	//-------------------------------------------------------------------------------------------------------------------------------------------
	30:	//--- WriteParameter Vel_I AllSegments
		diResultSercosWriteServiceData 	:= SercosWriteServiceDataToAllSegments(	i_dwIDN					:= dwIDNCarrierVelI, 
																				i_dwDataStraightSegment	:= dwVelI_Straight, 
																				i_dwDataCurveSegment	:= dwVelI_Curve,
																				i_wMaxDataLength		:= 4);
		IF diResultSercosWriteServiceData = 0 THEN
			q_xWriteParameterDone	:= TRUE;
			diState	:= 40;
		ELSE
			q_xWriteParameterError	:= TRUE;
			diState	:= 1000;
		END_IF	
		
	//-------------------------------------------------------------------------------------------------------------------------------------------
	40: //--- WriteParameter TrackingDeviation WarningLevel AllSegments
		IF dwIDNDeviationLevelWarning > 0 THEN //--- value of 0 deactivate TrackingDeviation Detection
			diResultSercosWriteServiceData := SercosWriteServiceDataToAllSegments( 	i_dwIDN 				:= dwIDNDeviationLevelWarning,
																					i_dwDataStraightSegment	:= dwDeviationLevelWarning,
																					i_dwDataCurveSegment	:= dwDeviationLevelWarning,
																					i_wMaxDataLength 		:= 4);
		END_IF
		IF diResultSercosWriteServiceData = 0 THEN
			diState := 50;
		ELSE
			q_xWriteParameterError	:= TRUE;
			diState := 1000;
		END_IF

	//-------------------------------------------------------------------------------------------------------------------------------------------
	50: //--- WriteParameter TrackingDeviation ErrorLevel AllSegments
		IF dwIDNDeviationLevelError > 0 THEN //--- value of 0 deactivate TrackingDeviation Detection
			diResultSercosWriteServiceData := SercosWriteServiceDataToAllSegments( 	i_dwIDN 				:= dwIDNDeviationLevelError,
																					i_dwDataStraightSegment	:= dwDeviationLevelError,
																					i_dwDataCurveSegment	:= dwDeviationLevelError,
																					i_wMaxDataLength 		:= 4);
		END_IF
		IF diResultSercosWriteServiceData = 0 THEN
			diState := 60;
		ELSE
			q_xWriteParameterError	:= TRUE;
			diState := 1000;
		END_IF		
		
	//-------------------------------------------------------------------------------------------------------------------------------------------
	60:	//--- WriteParameter: Maximum Current AllSegments
		diResultSercosWriteServiceData 	:= SercosWriteServiceDataToAllSegments(	i_dwIDN					:= dwIDNCarrierMaxcurr, 
																				i_dwDataStraightSegment	:= dwMaxCurr, 
																				i_dwDataCurveSegment	:= dwMaxCurr,
																				i_wMaxDataLength		:= 2);
		IF diResultSercosWriteServiceData = 0 THEN
			diState := 70;
		ELSE
			q_xWriteParameterError	:= TRUE;
			diState	:= 1000;
		END_IF	
	
	//-------------------------------------------------------------------------------------------------------------------------------------------
	70:	//--- WriteParameter: Load of Carrier AllSegments
		diResultSercosWriteServiceData 	:= SercosWriteServiceDataToAllSegments(	i_dwIDN					:= dwIDNCarrierLoad, 
																				i_dwDataStraightSegment	:= dwMaxload, 
																				i_dwDataCurveSegment	:= dwMaxload, 
																				i_wMaxDataLength		:= 4);
		IF diResultSercosWriteServiceData = 0 THEN
			q_xWriteParameterDone	:= TRUE;
			diState := 0;
		ELSE
			q_xWriteParameterError	:= TRUE;
			diState	:= 1000;
		END_IF	
	
	//-------------------------------------------------------------------------------------------------------------------------------------------
	1000: //--- ErrorState
		;
	
END_CASE

METHOD SercosWriteServiceDataToAllSegments : DINT
VAR_INPUT
	i_dwIDN					: DWORD;
	i_dwDataCurveSegment	: DWORD;	
	i_dwDataStraightSegment	: DWORD;	
	i_wMaxDataLength		: WORD;
END_VAR
VAR
	udiIndex				: UDINT;
END_VAR
FOR udiIndex := 1  TO GVL_MulticarrierConfiguration.Gc_astTracks[1].udiNumberOfSegments DO
	

    IF GVL_MulticarrierConfiguration.Gc_astSegmentTypes[GVL_MulticarrierConfiguration.Gc_astTracks[1].astSegments[udiIndex].diSegmentTypesIndex].xIsCurved  
    THEN        
        SercosWriteServiceDataToAllSegments := SystemInterface.FC_SercosWriteServiceDataByTopAddr(    
                                                                    i_wTopoAddr         := TO_WORD(udiIndex), 
                                                                    i_dwIDN             := i_dwIDN,
                                                                    i_wType             := 5,
                                                                    i_dwPointerToData   := ADR(i_dwDataCurveSegment),
                                                                    i_wMaxDataLen       := i_wMaxDataLength);
    ELSE
        SercosWriteServiceDataToAllSegments := SystemInterface.FC_SercosWriteServiceDataByTopAddr(    
                                                                    i_wTopoAddr         := TO_WORD(udiIndex), 
                                                                    i_dwIDN             := i_dwIDN,
                                                                    i_wType             := 5,
                                                                    i_dwPointerToData   := ADR(i_dwDataStraightSegment),
                                                                    i_wMaxDataLen       := i_wMaxDataLength);
    END_IF    

    IF SercosWriteServiceDataToAllSegments <> 0 THEN
        RETURN;
    END_IF
END_FOR
END_METHOD

METHOD StartAndSetParameter
VAR_INPUT
	i_dwPosP_Straight				: DWORD;
	i_dwVelP_Straight				: DWORD;
	i_dwVelI_Straight				: DWORD;  
	i_dwPosP_Curve					: DWORD;
	i_dwVelP_Curve					: DWORD;
	i_dwVelI_Curve					: DWORD;  
	i_dwMaxCurr			            : DWORD;
    i_dwMaxload					    : DWORD;
    i_dwDeviationLevelWarning       : DWORD;
    i_dwDeviationLevelError         : DWORD;
	
	
	
END_VAR
dwPosP_Straight	:= 	i_dwPosP_Straight;
dwVelP_Straight	:=	i_dwVelP_Straight;
dwVelI_Straight	:=	i_dwVelI_Straight;

dwPosP_Curve	:= 	i_dwPosP_Curve;
dwVelP_Curve	:=	i_dwVelP_Curve;
dwVelI_Curve	:=	i_dwVelI_Curve;

dwMaxCurr			      := i_dwMaxCurr;
dwMaxload				  := i_dwMaxload;
dwDeviationLevelWarning   := i_dwDeviationLevelWarning;
dwDeviationLevelError     := i_dwDeviationLevelError;

xStart 		:=  TRUE;
END_METHOD

END_PROGRAM

// LMC_PacDrive/Application/TemplateFullProgrammingFramework/TaskCalls/SR_Diagnostics
PROGRAM SR_Diagnostics

VAR
	fbDiagnosticsManager : TPL.FB_DiagnosticsManager;
	stComStructure 		 : TPL.ST_DiagnosticsManagerToDiagSource;
	
	stWarning 		: TPL.ST_Exception;
	etLastDiagExt	: TPL.ET_DiagExt := TPL.ET_DiagExt.Ok;

	(* Add the instances of your sources for diag data here *)
	fbTemplateStaticStructureDiagSource	: TPL.FB_TemplateStaticStructureDiagSource;
	fbExceptionListDiagSource			: TPL.FB_ExceptionListDiagSource;
	fbExceptionDelayListDiagSource		: TPL.FB_ExceptionDelayListDiagSource;
	fbLogDataListDiagSource				: TPL.FB_LogDataListDiagSource;	
	fbAxisModuleDiagSource				: AXM.FB_AxisModuleDiagSource;
	xPrintCamData						: BOOL := TRUE;
	fbApplicationLoggerDiagSource		: FB_ApplicationLoggerDiagSource;

	(* example diag sources *)
	fbExampleTableDiagSource			: FB_ExampleTableDiagSource;
	fbExampleTreeDiagSource				: FB_ExampleTreeDiagSource;
END_VAR

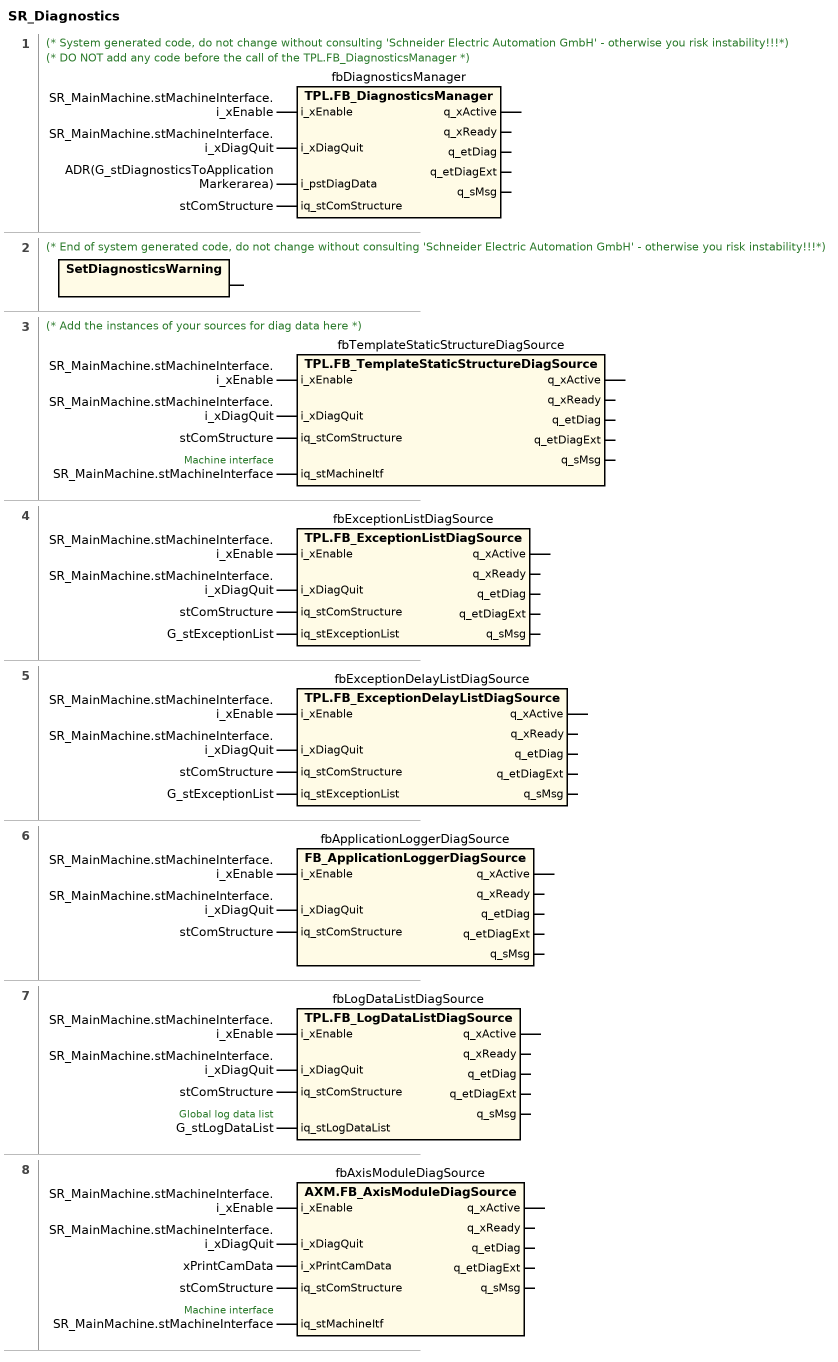
// NETWORK 1
// (* System generated code, do not change without consulting 'Schneider Electric Automation GmbH' - otherwise you risk instability!!!*)
// (* DO NOT add any code before the call of the TPL.FB_DiagnosticsManager *)
fbDiagnosticsManager(
    i_xEnable := SR_MainMachine.stMachineInterface.i_xEnable,
    i_xDiagQuit := SR_MainMachine.stMachineInterface.i_xDiagQuit,
    i_pstDiagData := ADR(G_stDiagnosticsToApplicationMarkerarea),
    iq_stComStructure := stComStructure); // TPL.FB_DiagnosticsManager

// NETWORK 2
// (* End of system generated code, do not change without consulting 'Schneider Electric Automation GmbH' - otherwise you risk instability!!!*)
SetDiagnosticsWarning();

// NETWORK 3
// (* Add the instances of your sources for diag data here *)
//   fbTemplateStaticStructureDiagSource: Add the instances of your sources for diag data here
//   SR_MainMachine.stMachineInterface: Machine interface
fbTemplateStaticStructureDiagSource(
    i_xEnable := SR_MainMachine.stMachineInterface.i_xEnable,
    i_xDiagQuit := SR_MainMachine.stMachineInterface.i_xDiagQuit,
    iq_stComStructure := stComStructure,
    iq_stMachineItf := SR_MainMachine.stMachineInterface); // TPL.FB_TemplateStaticStructureDiagSource

// NETWORK 4
fbExceptionListDiagSource(
    i_xEnable := SR_MainMachine.stMachineInterface.i_xEnable,
    i_xDiagQuit := SR_MainMachine.stMachineInterface.i_xDiagQuit,
    iq_stComStructure := stComStructure,
    iq_stExceptionList := G_stExceptionList); // TPL.FB_ExceptionListDiagSource

// NETWORK 5
fbExceptionDelayListDiagSource(
    i_xEnable := SR_MainMachine.stMachineInterface.i_xEnable,
    i_xDiagQuit := SR_MainMachine.stMachineInterface.i_xDiagQuit,
    iq_stComStructure := stComStructure,
    iq_stExceptionList := G_stExceptionList); // TPL.FB_ExceptionDelayListDiagSource

// NETWORK 6
fbApplicationLoggerDiagSource(
    i_xEnable := SR_MainMachine.stMachineInterface.i_xEnable,
    i_xDiagQuit := SR_MainMachine.stMachineInterface.i_xDiagQuit,
    iq_stComStructure := stComStructure); // FB_ApplicationLoggerDiagSource

// NETWORK 7
//   G_stLogDataList: Global log data list
fbLogDataListDiagSource(
    i_xEnable := SR_MainMachine.stMachineInterface.i_xEnable,
    i_xDiagQuit := SR_MainMachine.stMachineInterface.i_xDiagQuit,
    iq_stComStructure := stComStructure,
    iq_stLogDataList := G_stLogDataList); // TPL.FB_LogDataListDiagSource

// NETWORK 8
//   SR_MainMachine.stMachineInterface: Machine interface
fbAxisModuleDiagSource(
    i_xEnable := SR_MainMachine.stMachineInterface.i_xEnable,
    i_xDiagQuit := SR_MainMachine.stMachineInterface.i_xDiagQuit,
    i_xPrintCamData := xPrintCamData,
    iq_stComStructure := stComStructure,
    iq_stMachineItf := SR_MainMachine.stMachineInterface); // AXM.FB_AxisModuleDiagSource

ACTION SetDiagnosticsWarning:
(* System generated code, do not change without consulting 'Schneider Electric Automation GmbH' - otherwise you risk instability!!!*)
						
(* Signal exception during diagnostics, but as diagnostics should not influence the machine, create only a warning *)
IF(fbDiagnosticsManager.q_etDiag <> GD.ET_Diag.Ok AND fbDiagnosticsManager.q_etDiagExt <> etLastDiagExt) THEN
	
	stWarning.etDiag		:= GD.ET_Diag.DiagActive;
	stWarning.udiDiagExt	:= ET_DiagExt.DiagnosticsWarning;
	stWarning.sDiagExt		:= FC_EtDiagExtToString(stWarning.udiDiagExt);
	stWarning.udiModuleId	:= SR_MainMachine.c_udiMainModuleId;
	stWarning.sMsg			:= CONCAT(CONCAT('SR_Diagnostics: ', GD.FC_EtDiagToString(fbDiagnosticsManager.q_etDiag)), CONCAT(' ; ', TPL.FC_EtDiagExtToString(fbDiagnosticsManager.q_etDiagExt)));
	stWarning.sModuleName	:= SR_MainMachine.stMachineInterface.i_sModuleName;
	stWarning.etSource		:= TPL.ET_ExceptionSource.Logger;
	
	TPL.FC_SetException(i_xExceptionActive	:= TRUE,
						iq_stException		:= stWarning,
						iq_stExceptionList	:= G_stExceptionList,
						iq_stLogDataList	:= G_stLogDataList);
END_IF

etLastDiagExt := fbDiagnosticsManager.q_etDiagExt;
(* End of system generated code, do not change without consulting 'Schneider Electric Automation GmbH' - otherwise you risk instability!!!*)
END_ACTION

END_PROGRAM

// LMC_PacDrive/Application/TemplateFullProgrammingFramework/Examples/ExampleDiagSources/FB_ApplicationLoggerDiagSource
FUNCTION_BLOCK PUBLIC FB_ApplicationLoggerDiagSource
VAR_INPUT
	i_xEnable			: BOOL;
	i_xDiagQuit			: BOOL;
END_VAR

VAR_IN_OUT
	iq_stComStructure	: TPL.ST_DiagnosticsManagerToDiagSource;
END_VAR

VAR_OUTPUT
	q_xActive			: BOOL;
	q_xReady			: BOOL;
	q_etDiag			: GD.ET_Diag := GD.ET_Diag.Ok;
	q_etDiagExt			: ET_DiagExt := ET_DiagExt.Disabled;
	q_sMsg				: STRING[80];
END_VAR

VAR
	xEnableFlag		: BOOL;
	diState			: DINT;

	udiOwnSourceId	: UDINT := 0;

	fbTreeWriter	: TPL.FB_TreeWriter;
	
	diOldCmd		: DINT := 0;
	diCmdExecState	: DINT := 0;

	etDiagBuffer		: GD.ET_Diag;
	etDiagExtBufferTPL	: TPL.ET_DiagExt;
	etDiagExtBufferAPL	: APL.ET_DiagExt;
	sMsgBuffer			: STRING[80];
	
	rtrigDiagQuit	: Standard.R_TRIG;
	
	fbAppLogHandler			: APL.FB_ApplicationLoggerHandler;
	stLogEntry				: APL.ST_LogEntry;
	ifLoggerPoint			: APL.IF_LoggerPoint;
	udiLogEntryCount		: UDINT;
	udiLogEntryCountMax		: UDINT;
	udiLogEntryId			: UDINT;
	udiLoggerPointCount		: UDINT;
	udiLoggerPointCountMax	: UDINT;
END_VAR

VAR CONSTANT
	c_sName			: STRING[TPL.Gc_udiTableWriterMaxNameLength] := 'ApplicationLogger';
	c_sTypeName		: STRING[TPL.Gc_udiTableWriterMaxNameLength] := 'APL_';
END_VAR

IF i_xEnable AND NOT xEnableFlag THEN
	xEnableFlag := TRUE;
	q_xActive := TRUE;
	SetDiagOutputs(	i_etDiag	:= GD.ET_Diag.Ok,
					i_etDiagExt	:= ET_DiagExt.WaitUntilDiagnosticsManagerReady,
					i_sMsg		:= '');	
	diState := 10;
	
ELSIF NOT i_xEnable AND xEnableFlag THEN
	xEnableFlag := FALSE;
	IF udiOwnSourceId <> 0 THEN		
		SetDiagOutputs(	i_etDiag	:= GD.ET_Diag.Ok,
						i_etDiagExt	:= ET_DiagExt.WaitUntilDisabled,
						i_sMsg		:= '');
		diState := 100;
	ELSIF udiOwnSourceId = 0 THEN		
		SetDiagOutputs(	i_etDiag	:= GD.ET_Diag.Ok,
						i_etDiagExt	:= ET_DiagExt.Disabled,
						i_sMsg		:= '');
	END_IF
END_IF

DiagQuit();

CASE diState OF
	
	0:	(* Disable & exception state *)
		;
	
	10:	(* Wait until diagnostics manager ready *)
		IF iq_stComStructure.i_xDiagnosticsManagerReady THEN
			SetDiagOutputs(	i_etDiag	:= GD.ET_Diag.Ok,
							i_etDiagExt	:= ET_DiagExt.WaitUntilDiagSourceRegistered,
							i_sMsg		:= '');
			diState := 20;
		END_IF

	20:	(* Wait until diag source registered *)	
		IF NOT iq_stComStructure.i_xDiagnosticsManagerReady THEN
			SetDiagOutputs(	i_etDiag	:= GD.ET_Diag.Ok,
							i_etDiagExt	:= ET_DiagExt.WaitUntilDiagnosticsManagerReady,
							i_sMsg		:= '');	
			diState := 10;
	
		(* only write to register structure if no one else has done it in this cylce *)
		ELSIF (NOT iq_stComStructure.iq_stRegister.xUsed AND iq_stComStructure.iq_stRegister.udiNextId <> 0) THEN
			(* register *)
			iq_stComStructure.iq_stRegister.xUsed := TRUE;
			iq_stComStructure.iq_stRegister.sName		:= c_sName;
			iq_stComStructure.iq_stRegister.sTypeName	:= c_sTypeName;
			udiOwnSourceId := iq_stComStructure.iq_stRegister.udiNextId; (* register with this id; required for the following communication *)
			
			q_xReady := TRUE;
			SetDiagOutputs(	i_etDiag	:= GD.ET_Diag.Ok,
							i_etDiagExt	:= ET_DiagExt.WaitForCommunication,
							i_sMsg		:= '');
			diState := 30;
		END_IF
	
	30:	(* Wait for communication *)	
		IF NOT iq_stComStructure.i_xDiagnosticsManagerReady THEN

			CancelWriting();
									
			udiOwnSourceId	:= 0;
			
			SetDiagOutputs(	i_etDiag	:= GD.ET_Diag.Ok,
							i_etDiagExt	:= ET_DiagExt.WaitUntilDiagnosticsManagerReady,
							i_sMsg		:= '');	
			diState := 10;
			RETURN;
			
		ELSIF (iq_stComStructure.i_udiComWithId = udiOwnSourceId) THEN		(* Am I adressed? *)
			
			WriteDiagDataControl();

		ELSE
			iq_stComStructure.q_lrProgress := 0.0;
			
			CancelWriting();
						
			SetDiagOutputs(	i_etDiag	:= GD.ET_Diag.Ok,
							i_etDiagExt	:= ET_DiagExt.WaitForCommunication,
							i_sMsg		:= '');
		END_IF
		
	100: (* Wait until disabled *)	
		IF NOT iq_stComStructure.i_xDiagnosticsManagerReady THEN

			CancelWriting();
									
			udiOwnSourceId	:= 0;
			
			SetDiagOutputs(	i_etDiag	:= GD.ET_Diag.Ok,
							i_etDiagExt	:= ET_DiagExt.Disabled,
							i_sMsg		:= '');	
	
		ELSIF (iq_stComStructure.i_udiComWithId = udiOwnSourceId) THEN		(* Am I adressed? *)
			
			WriteDiagDataControl();
			
		(* only write to register structure if no one else has done it in this cylce *)
		ELSIF (NOT iq_stComStructure.iq_stRegister.xUsed AND NOT iq_stComStructure.iq_stRegister.xUnsubscribe) AND 
			   NOT iq_stComStructure.i_xDiagnosticsActive THEN
			   
			iq_stComStructure.iq_stRegister.xUsed			:= TRUE;
			
			iq_stComStructure.iq_stRegister.xUnsubscribe	:= TRUE;
			iq_stComStructure.iq_stRegister.udiSourceId		:= udiOwnSourceId;
			
			q_xActive := FALSE;
			
			SetDiagOutputs(	i_etDiag	:= GD.ET_Diag.Ok,
							i_etDiagExt	:= ET_DiagExt.Disabled,
							i_sMsg		:= '');
		END_IF
END_CASE

IF q_xReady THEN	
	IF(diCmdExecState <> 0) THEN
		WriteDiagDataToFile();
		
		IF(iq_stComStructure.iq_diCmd <= 0) THEN
			diOldCmd := iq_stComStructure.iq_diCmd;
		END_IF
	END_IF	
END_IF

METHOD INTERNAL CancelWriting
VAR_INPUT
END_VAR
(* Deactivate writing if we are (for whatever reason) no longer adressed.
   May happen in case network connection with Diagnostics is disrupted or Source will be disabled *)

THIS^.diOldCmd			:= 0;
THIS^.diCmdExecState	:= 0;
END_METHOD

METHOD INTERNAL DiagQuit
VAR_INPUT
END_VAR
IF THIS^.i_xEnable AND THIS^.q_xActive AND THIS^.q_etDiag <> GD.ET_Diag.Ok AND THIS^.diState = 0 THEN

	THIS^.rtrigDiagQuit(CLK := THIS^.i_xDiagQuit);
	IF THIS^.rtrigDiagQuit.Q THEN
		CancelWriting();
									
		THIS^.udiOwnSourceId	:= 0;
		
		THIS^.fbTreeWriter.FB_Init(bInitRetains := FALSE, bInCopyCode := FALSE);
			
		THIS^.q_xReady		:= TRUE;
		THIS^.q_etDiag		:= GD.ET_Diag.Ok;
		THIS^.q_etDiagExt	:= ET_DiagExt.WaitUntilDiagnosticsManagerReady;
		THIS^.q_sMsg		:= '';
	
		THIS^.diState := 10;
	END_IF

END_IF
END_METHOD

METHOD INTERNAL ExceptionDuringWriting : BOOL
VAR_INPUT
END_VAR
(* exception during writing *)
CASE THIS^.etDiagExtBufferTPL OF
	TPL.ET_DiagExt.TreeStartAlreadySuccessfullyCalled,		// FB_TreeWriter.TreeStart	
	TPL.ET_DiagExt.FileIdNotSet,							// FB_TreeWriter.TreeStart							
	TPL.ET_DiagExt.FileIdInvalid,							// FB_TreeWriter.TreeStart & FB_TreeWriter.NodeStart & FB_TreeWriter.Parameter & FB_TreeWriter.NodeEnd & FB_TreeWriter.TreeEnd								
	TPL.ET_DiagExt.FileNotOpen,								// FB_TreeWriter.TreeStart & FB_TreeWriter.NodeStart & FB_TreeWriter.Parameter & FB_TreeWriter.NodeEnd & FB_TreeWriter.TreeEnd								
	TPL.ET_DiagExt.UnexpectedFeedback,						// FB_TreeWriter.TreeStart & FB_TreeWriter.NodeStart & FB_TreeWriter.Parameter & FB_TreeWriter.NodeEnd & FB_TreeWriter.TreeEnd								
	TPL.ET_DiagExt.TreeStartNotCalled,						// FB_TreeWriter.NodeStart								
	TPL.ET_DiagExt.TreeStartNotSuccessfullyCalled,			// FB_TreeWriter.NodeStart								
	TPL.ET_DiagExt.NoMoreNodeOpen,							// FB_TreeWriter.Parameter & FB_TreeWriter.NodeEnd						
	TPL.ET_DiagExt.CallTreeStartFirst,						// FB_TreeWriter.TreeEnd								
	TPL.ET_DiagExt.NodesStillOpen:							// FB_TreeWriter.TreeEnd	
	
		SetDiagOutputs(	i_etDiag	:= GD.ET_Diag.UnexpectedProgramBehavior,
						i_etDiagExt	:= ET_DiagExt.UnexpectedFeedback,
						i_sMsg		:= PDL.FC_MultiConcat(	i_sString1	:= 'FB_TreeWriter: ', 
															i_sString2	:= GD.FC_EtDiagToString(THIS^.etDiagBuffer), 
															i_sString3	:= ' - ', 
															i_sString4	:= TPL.FC_EtDiagExtToString(THIS^.etDiagExtBufferTPL), 
															q_etDiag	=> , 
															q_etDiagExt	=> )); 								
	ELSE
		SetDiagOutputs(	i_etDiag	:= GD.ET_Diag.UnexpectedProgramBehavior,
						i_etDiagExt	:= ET_DiagExt.UnexpectedFeedback,
						i_sMsg		:= PDL.FC_MultiConcat(	i_sString1	:= 'FB_TreeWriter: ', 
															i_sString2	:= GD.FC_EtDiagToString(THIS^.etDiagBuffer), 
															i_sString3	:= ' - ', 
															i_sString4	:= TPL.FC_EtDiagExtToString(THIS^.etDiagExtBufferTPL), 
															q_etDiag	=> , 
															q_etDiagExt	=> )); 						
END_CASE
		
CancelWriting();
END_METHOD

METHOD INTERNAL SetDiagOutputs : BOOL
VAR_INPUT
	i_etDiag		: GD.ET_Diag;
	i_etDiagExt		: ET_DiagExt;
	i_sMsg			: STRING[80];
END_VAR
IF THIS^.q_etDiag = GD.ET_Diag.Ok OR i_etDiagExt = ET_DiagExt.Disabled THEN

	IF i_etDiag <> GD.ET_Diag.Ok OR i_etDiagExt = ET_DiagExt.Disabled THEN
		
		IF i_etDiag <> GD.ET_Diag.Ok THEN
			THIS^.iq_stComStructure.iq_diCmd := -THIS^.iq_stComStructure.iq_diCmd;
		END_IF
		
		IF i_etDiagExt = ET_DiagExt.Disabled THEN
			THIS^.q_xActive := FALSE;
			
			CancelWriting();
		END_IF
		
		THIS^.q_xReady := FALSE;
		THIS^.diState := 0;
	END_IF
	
	THIS^.q_etDiag		:= i_etDiag;
	THIS^.q_etDiagExt	:= i_etDiagExt;
	THIS^.q_sMsg		:= i_sMsg;
END_IF
END_METHOD

METHOD INTERNAL WriteDiagDataControl : BOOL
VAR_INPUT
END_VAR
IF (THIS^.diOldCmd <> THIS^.iq_stComStructure.iq_diCmd AND THIS^.iq_stComStructure.iq_diCmd > 0) THEN
	THIS^.diOldCmd := THIS^.iq_stComStructure.iq_diCmd;
	
	(* new command, start execution *)
	IF THIS^.iq_stComStructure.iq_diCmd = 1 THEN
		IF (THIS^.iq_stComStructure.i_diFileId > 0) THEN
			SetDiagOutputs(	i_etDiag		:= GD.ET_Diag.Ok,
							i_etDiagExt		:= ET_DiagExt.WritingToFile,
							i_sMsg			:= '');
			THIS^.iq_stComStructure.q_lrProgress := 0.0;
			THIS^.fbTreeWriter.diFileId := THIS^.iq_stComStructure.i_diFileId;
			THIS^.diCmdExecState := 1; (* start writing to file *)
		ELSE
			(* invalid file id *)
			SetDiagOutputs(	i_etDiag		:= GD.ET_Diag.InputParameterInvalid,
							i_etDiagExt		:= ET_DiagExt.FileIdInvalid,
							i_sMsg			:= CONCAT('Invalid file Id iq_stComStructure.i_diFileId: ', DINT_TO_STRING(THIS^.iq_stComStructure.i_diFileId)));
		END_IF
	ELSE
		(* unkown cmd *)
		SetDiagOutputs(	i_etDiag		:= GD.ET_Diag.InputParameterInvalid,
						i_etDiagExt		:= ET_DiagExt.CmdUnknown,
						i_sMsg			:= CONCAT('Unknown command iq_stComStructure.diCmd: ', DINT_TO_STRING(THIS^.iq_stComStructure.iq_diCmd)));

		CancelWriting();
	END_IF
END_IF
END_METHOD

METHOD WriteDiagDataToFile
VAR_INPUT
END_VAR
TPL.FC_CanContinueWriting(iq_stCanContinueWriting := THIS^.iq_stComStructure.iq_stCanContinueWriting); (* loop as long as we can continue to write *)

WHILE (THIS^.iq_stComStructure.iq_stCanContinueWriting.xCanContinue) DO
	
	CASE THIS^.diCmdExecState OF
		1:	(* start writing *)
			THIS^.fbTreeWriter.TreeStart(	i_sName					:= THIS^.c_sName, 
											i_sTypeName				:= THIS^.c_sTypeName, 
											i_sTitleEnglish			:= 'ApplicationLogger', 
											i_sTitleGerman			:= 'ApplicationLogger', 
											i_uiPrintRank			:= 14, 
											i_sEmptyListTextEnglish	:= 'No data available to show', 
											i_sEmptyListTextGerman	:= 'Keine Daten zum Anzeigen vorhanden',
											q_etDiag				=> THIS^.etDiagBuffer,
											q_etDiagExt				=> THIS^.etDiagExtBufferTPL,
											q_sMsg					=> THIS^.sMsgBuffer);
			IF THIS^.etDiagBuffer <> GD.ET_Diag.Ok THEN
				ExceptionDuringWriting();
				EXIT;
			END_IF
			THIS^.diCmdExecState := 50;

		50:	(* Start LogEntryList *)
			THIS^.fbTreeWriter.NodeStart(	i_sName		:= 'LogEntry list',
											q_etDiag	=> etDiagBuffer,
											q_etDiagExt	=> etDiagExtBufferTPL,
											q_sMsg		=> sMsgBuffer);
			IF THIS^.etDiagBuffer <> GD.ET_Diag.Ok THEN
				ExceptionDuringWriting();
				EXIT;
			END_IF
			THIS^.udiLogEntryCount := 1;
			THIS^.udiLogEntryCountMax := 50;
			THIS^.udiLogEntryId := THIS^.fbAppLogHandler.udiFirstLogEntryId;
			THIS^.diCmdExecState := 51;
			
		51: (* write LogEntrys *)
			WHILE (THIS^.udiLogEntryCount < THIS^.udiLogEntryCountMax) AND (THIS^.udiLogEntryCount <= THIS^.fbAppLogHandler.udiNumberOfLogEntries) DO
				THIS^.fbTreeWriter.NodeStart(	i_sName		:= UDINT_TO_STRING(THIS^.udiLogEntryId),
												q_etDiag	=> etDiagBuffer,
												q_etDiagExt	=> etDiagExtBufferTPL,
												q_sMsg		=> sMsgBuffer);
				IF THIS^.etDiagBuffer <> GD.ET_Diag.Ok THEN
					ExceptionDuringWriting();
					RETURN;
				END_IF					

					THIS^.fbAppLogHandler.GetLogEntry(	i_udiId			:= THIS^.udiLogEntryId,
														q_stLogEntry	=> THIS^.stLogEntry,
														q_etDiag		=> THIS^.etDiagBuffer,
														q_etDiagExt		=> THIS^.etDiagExtBufferAPL);
					IF (THIS^.etDiagBuffer <> GD.ET_Diag.Ok) THEN
						ExceptionDuringWriting();
						RETURN;
					END_IF
				
					THIS^.fbTreeWriter.Parameter(	i_sName		:= 'udiId', 
													i_sValue	:= UDINT_TO_STRING(THIS^.stLogEntry.udiId),
													q_etDiag	=> etDiagBuffer,
													q_etDiagExt	=> etDiagExtBufferTPL,
													q_sMsg		=> sMsgBuffer);
					IF etDiagBuffer <> GD.ET_Diag.Ok THEN
						ExceptionDuringWriting();
						RETURN;
					END_IF

					THIS^.fbTreeWriter.Parameter(	i_sName		:= 'udiLoggerPointId', 
													i_sValue	:= UDINT_TO_STRING(THIS^.stLogEntry.udiLoggerPointId),
													q_etDiag	=> etDiagBuffer,
													q_etDiagExt	=> etDiagExtBufferTPL,
													q_sMsg		=> sMsgBuffer);
					IF etDiagBuffer <> GD.ET_Diag.Ok THEN
						ExceptionDuringWriting();
						RETURN;
					END_IF
					THIS^.fbTreeWriter.Parameter(	i_sName		:= 'sMessage', 
													i_sValue	:= THIS^.stLogEntry.sMessage,
													q_etDiag	=> etDiagBuffer,
													q_etDiagExt	=> etDiagExtBufferTPL,
													q_sMsg		=> sMsgBuffer);
					IF etDiagBuffer <> GD.ET_Diag.Ok THEN
						ExceptionDuringWriting();
						RETURN;
					END_IF
					THIS^.fbTreeWriter.Parameter(	i_sName		:= 'etDiag', 
													i_sValue	:= GD.FC_EtDiagToString(i_etDiag := THIS^.stLogEntry.etDiag),
													q_etDiag	=> etDiagBuffer,
													q_etDiagExt	=> etDiagExtBufferTPL,
													q_sMsg		=> sMsgBuffer);
					IF etDiagBuffer <> GD.ET_Diag.Ok THEN
						ExceptionDuringWriting();
						RETURN;
					END_IF
					THIS^.fbTreeWriter.Parameter(	i_sName		:= 'udiDiagExt', 
													i_sValue	:= UDINT_TO_STRING(THIS^.stLogEntry.udiDiagExt),
													q_etDiag	=> etDiagBuffer,
													q_etDiagExt	=> etDiagExtBufferTPL,
													q_sMsg		=> sMsgBuffer);
					IF etDiagBuffer <> GD.ET_Diag.Ok THEN
						ExceptionDuringWriting();
						RETURN;
					END_IF
					THIS^.fbTreeWriter.Parameter(	i_sName		:= 'dtDate', 
													i_sValue	:= DATE_TO_STRING(THIS^.stLogEntry.dtDate),
													q_etDiag	=> etDiagBuffer,
													q_etDiagExt	=> etDiagExtBufferTPL,
													q_sMsg		=> sMsgBuffer);
					IF etDiagBuffer <> GD.ET_Diag.Ok THEN
						ExceptionDuringWriting();
						RETURN;
					END_IF
					THIS^.fbTreeWriter.Parameter(	i_sName		:= 'todTime', 
													i_sValue	:= TOD_TO_STRING(THIS^.stLogEntry.todTime),
													q_etDiag	=> etDiagBuffer,
													q_etDiagExt	=> etDiagExtBufferTPL,
													q_sMsg		=> sMsgBuffer);
					IF etDiagBuffer <> GD.ET_Diag.Ok THEN
						ExceptionDuringWriting();
						RETURN;
					END_IF
					THIS^.fbTreeWriter.Parameter(	i_sName		:= 'etLogLevel', 
													i_sValue	:= APL.FC_EtLogLevelToString(i_etLogLevel := THIS^.stLogEntry.etLogLevel),
													q_etDiag	=> etDiagBuffer,
													q_etDiagExt	=> etDiagExtBufferTPL,
													q_sMsg		=> sMsgBuffer);
					IF etDiagBuffer <> GD.ET_Diag.Ok THEN
						ExceptionDuringWriting();
						RETURN;
					END_IF
					
				THIS^.fbTreeWriter.NodeEnd(	q_etDiag	=> etDiagBuffer,
											q_etDiagExt	=> etDiagExtBufferTPL,
											q_sMsg		=> sMsgBuffer);	
				IF THIS^.etDiagBuffer <> GD.ET_Diag.Ok THEN
					ExceptionDuringWriting();
					RETURN;
				END_IF	
			
				THIS^.udiLogEntryCount := THIS^.udiLogEntryCount +1;
				THIS^.udiLogEntryId := THIS^.udiLogEntryId +1;
			END_WHILE
			THIS^.udiLogEntryCountMax := THIS^.udiLogEntryCountMax + 50;
			IF (THIS^.udiLogEntryCount > THIS^.fbAppLogHandler.udiNumberOfLogEntries) THEN
				THIS^.fbTreeWriter.NodeEnd(	q_etDiag	=> etDiagBuffer,
											q_etDiagExt	=> etDiagExtBufferTPL,
											q_sMsg		=> sMsgBuffer);	
				IF THIS^.etDiagBuffer <> GD.ET_Diag.Ok THEN
					ExceptionDuringWriting();
					EXIT;
				END_IF
				THIS^.diCmdExecState := 60;
			END_IF
		
		60: (* Start LoggerPoint list *)
			THIS^.fbTreeWriter.NodeStart(	i_sName		:= 'LoggerPoint list',
											q_etDiag	=> etDiagBuffer,
											q_etDiagExt	=> etDiagExtBufferTPL,
											q_sMsg		=> sMsgBuffer);
			IF THIS^.etDiagBuffer <> GD.ET_Diag.Ok THEN
				ExceptionDuringWriting();
				EXIT;
			END_IF
			THIS^.udiLoggerPointCount := 1;
			THIS^.udiLoggerPointCountMax := 50;
			THIS^.diCmdExecState := 61;	
			
		61: (* write LoggerPoint list *)
			WHILE (THIS^.udiLoggerPointCount < THIS^.udiLoggerPointCountMax) AND (THIS^.udiLoggerPointCount <= THIS^.fbAppLogHandler.udiNumberOfLoggerPoints) DO
				THIS^.fbTreeWriter.NodeStart(	i_sName		:= UDINT_TO_STRING(THIS^.udiLoggerPointCount),
												q_etDiag	=> etDiagBuffer,
												q_etDiagExt	=> etDiagExtBufferTPL,
												q_sMsg		=> sMsgBuffer);
				IF THIS^.etDiagBuffer <> GD.ET_Diag.Ok THEN
					ExceptionDuringWriting();
					RETURN;
				END_IF					

					THIS^.fbAppLogHandler.GetLoggerPoint(	i_udiId			:= THIS^.udiLoggerPointCount,
															q_ifLoggerPoint	=> THIS^.ifLoggerPoint,
															q_etDiag		=> THIS^.etDiagBuffer,
															q_etDiagExt		=> THIS^.etDiagExtBufferAPL);
					IF (THIS^.etDiagBuffer <> GD.ET_Diag.Ok) THEN
						ExceptionDuringWriting();
						RETURN;
					END_IF
				
					THIS^.fbTreeWriter.Parameter(	i_sName		:= 'udiId', 
													i_sValue	:= UDINT_TO_STRING(THIS^.ifLoggerPoint.udiId),
													q_etDiag	=> etDiagBuffer,
													q_etDiagExt	=> etDiagExtBufferTPL,
													q_sMsg		=> sMsgBuffer);
					IF etDiagBuffer <> GD.ET_Diag.Ok THEN
						ExceptionDuringWriting();
						RETURN;
					END_IF			
					THIS^.fbTreeWriter.Parameter(	i_sName		:= 'udiParentId', 
													i_sValue	:= UDINT_TO_STRING(THIS^.ifLoggerPoint.udiParentId),
													q_etDiag	=> etDiagBuffer,
													q_etDiagExt	=> etDiagExtBufferTPL,
													q_sMsg		=> sMsgBuffer);
					IF etDiagBuffer <> GD.ET_Diag.Ok THEN
						ExceptionDuringWriting();
						RETURN;
					END_IF
					THIS^.fbTreeWriter.Parameter(	i_sName		:= 'sName', 
													i_sValue	:= THIS^.ifLoggerPoint.sName,
													q_etDiag	=> etDiagBuffer,
													q_etDiagExt	=> etDiagExtBufferTPL,
													q_sMsg		=> sMsgBuffer);
					IF etDiagBuffer <> GD.ET_Diag.Ok THEN
						ExceptionDuringWriting();
						RETURN;
					END_IF			
					THIS^.fbTreeWriter.Parameter(	i_sName		:= 'sType', 
													i_sValue	:= THIS^.ifLoggerPoint.sType,
													q_etDiag	=> etDiagBuffer,
													q_etDiagExt	=> etDiagExtBufferTPL,
													q_sMsg		=> sMsgBuffer);
					IF etDiagBuffer <> GD.ET_Diag.Ok THEN
						ExceptionDuringWriting();
						RETURN;
					END_IF
					THIS^.fbTreeWriter.Parameter(	i_sName		:= 'sSource', 
													i_sValue	:= THIS^.ifLoggerPoint.sSource,
													q_etDiag	=> etDiagBuffer,
													q_etDiagExt	=> etDiagExtBufferTPL,
													q_sMsg		=> sMsgBuffer);
					IF etDiagBuffer <> GD.ET_Diag.Ok THEN
						ExceptionDuringWriting();
						RETURN;
					END_IF
					THIS^.fbTreeWriter.Parameter(	i_sName		:= 'etLogLevel', 
													i_sValue	:= APL.FC_EtLogLevelToString(i_etLogLevel := THIS^.ifLoggerPoint.etLogLevel),
													q_etDiag	=> etDiagBuffer,
													q_etDiagExt	=> etDiagExtBufferTPL,
													q_sMsg		=> sMsgBuffer);
					IF etDiagBuffer <> GD.ET_Diag.Ok THEN
						ExceptionDuringWriting();
						RETURN;
					END_IF
			
				THIS^.fbTreeWriter.NodeEnd(	q_etDiag	=> etDiagBuffer,
											q_etDiagExt	=> etDiagExtBufferTPL,
											q_sMsg		=> sMsgBuffer);	
				IF THIS^.etDiagBuffer <> GD.ET_Diag.Ok THEN
					ExceptionDuringWriting();
					RETURN;
				END_IF	
			
				THIS^.udiLoggerPointCount := THIS^.udiLoggerPointCount +1;
			END_WHILE
			THIS^.udiLoggerPointCountMax := THIS^.udiLoggerPointCountMax + 50;
			IF (THIS^.udiLoggerPointCount > THIS^.fbAppLogHandler.udiNumberOfLoggerPoints) THEN
				THIS^.fbTreeWriter.NodeEnd(	q_etDiag	=> etDiagBuffer,
											q_etDiagExt	=> etDiagExtBufferTPL,
											q_sMsg		=> sMsgBuffer);	
				IF THIS^.etDiagBuffer <> GD.ET_Diag.Ok THEN
					ExceptionDuringWriting();
					EXIT;
				END_IF
				THIS^.diCmdExecState := 70;
			END_IF			
		
		70:
			(* library versions *)
			THIS^.fbTreeWriter.NodeStart(	i_sName		:= 'LibraryVersions',
											q_etDiag	=> THIS^.etDiagBuffer,
											q_etDiagExt	=> THIS^.etDiagExtBufferTPL,
											q_sMsg		=> THIS^.sMsgBuffer);				
			IF THIS^.etDiagBuffer <> GD.ET_Diag.Ok THEN
				ExceptionDuringWriting();
				EXIT;
			END_IF
			
				THIS^.fbTreeWriter.Parameter(	i_sName		:= 'ApplicationLogger', 
												i_sValue	:= APL.Gc_sLibraryVersion,
												q_etDiag	=> THIS^.etDiagBuffer,
												q_etDiagExt	=> THIS^.etDiagExtBufferTPL,
												q_sMsg		=> THIS^.sMsgBuffer);
				IF THIS^.etDiagBuffer <> GD.ET_Diag.Ok THEN
					ExceptionDuringWriting();
					EXIT;
				END_IF
			
				THIS^.fbTreeWriter.Parameter(	i_sName		:= 'GlobalDiagnostics', 
												i_sValue	:= GD.Gc_sLibraryVersion,
												q_etDiag	=> THIS^.etDiagBuffer,
												q_etDiagExt	=> THIS^.etDiagExtBufferTPL,
												q_sMsg		=> THIS^.sMsgBuffer);
				IF THIS^.etDiagBuffer <> GD.ET_Diag.Ok THEN
					ExceptionDuringWriting();
					EXIT;
				END_IF
				
			THIS^.fbTreeWriter.NodeEnd(	q_etDiag	=> THIS^.etDiagBuffer,
										q_etDiagExt	=> THIS^.etDiagExtBufferTPL,
										q_sMsg		=> THIS^.sMsgBuffer);		
			IF THIS^.etDiagBuffer <> GD.ET_Diag.Ok THEN
				ExceptionDuringWriting();
				EXIT;
			END_IF

			THIS^.fbTreeWriter.TreeEnd(	q_etDiag	=> THIS^.etDiagBuffer,
										q_etDiagExt	=> THIS^.etDiagExtBufferTPL,
										q_sMsg		=> THIS^.sMsgBuffer);	
			IF THIS^.etDiagBuffer <> GD.ET_Diag.Ok THEN
				ExceptionDuringWriting();
				EXIT;
			END_IF
			(* done *)
			
			(* signal command execution *)
			THIS^.iq_stComStructure.iq_diCmd := 0;
			
			SetDiagOutputs(	i_etDiag	:= GD.ET_Diag.Ok,
							i_etDiagExt	:= ET_DiagExt.DataSuccessfullyWritten,
							i_sMsg		:= '');		
			
			THIS^.diCmdExecState := 0;
			EXIT; (* exit the while loop *)
		ELSE
			ExceptionDuringWriting();
			EXIT;
	END_CASE
END_WHILE
END_METHOD

END_FUNCTION_BLOCK

// LMC_PacDrive/Application/TemplateFullProgrammingFramework/Examples/ExampleDiagSources/FB_ExampleTableDiagSource
FUNCTION_BLOCK FB_ExampleTableDiagSource
VAR_INPUT
	i_xEnable			: BOOL;
	i_xDiagQuit			: BOOL;
END_VAR

VAR_IN_OUT
	iq_stComStructure	: TPL.ST_DiagnosticsManagerToDiagSource;
END_VAR

VAR_OUTPUT
	q_xActive			: BOOL;
	q_xReady			: BOOL;
	q_etDiag			: GD.ET_Diag := GD.ET_Diag.Ok;
	q_etDiagExt			: ET_DiagExt := ET_DiagExt.Disabled;
	q_sMsg				: STRING[80];
END_VAR

VAR
	xEnableFlag		: BOOL;
	diState			: DINT;
	
	udiOwnSourceId : UDINT := 0;

	diOldCmd	: DINT := 0;
	diCmdExecState : DINT := 0;
	
	fbTableWriter : TPL.FB_TableWriter;

	udiCName : UDINT;
	udiCValue : UDINT;
	udiCC3 : UDINT;

	udiRowCounter : UDINT := 1;
	
	etDiag			: GD.ET_Diag;
	etDiagExtTPL	: TPL.ET_DiagExt;
	sMsg			: STRING[80];
	
	rtrigDiagQuit	: Standard.R_TRIG;
END_VAR

VAR CONSTANT
	c_sName : STRING[TPL.Gc_udiTableWriterMaxNameLength] := 'I_am_something';
	c_sTypeName : STRING[TPL.Gc_udiTableWriterMaxNameLength] := 'ExampleTableDiagSource';
	c_udiMaxNumRows : UDINT := 40;
END_VAR

IF i_xEnable AND NOT xEnableFlag THEN
	xEnableFlag := TRUE;
	
	q_xActive := TRUE;
	
	SetDiagOutputs(	i_etDiag	:= GD.ET_Diag.Ok,
					i_etDiagExt	:= ET_DiagExt.WaitUntilDiagnosticsManagerReady,
					i_sMsg		:= '');	
	diState := 10;
	
ELSIF NOT i_xEnable AND xEnableFlag THEN
	xEnableFlag := FALSE;
		
	IF udiOwnSourceId <> 0 THEN		
		SetDiagOutputs(	i_etDiag	:= GD.ET_Diag.Ok,
						i_etDiagExt	:= ET_DiagExt.WaitUntilDisabled,
						i_sMsg		:= '');
		diState := 100;
		
	ELSIF udiOwnSourceId = 0 THEN		
		SetDiagOutputs(	i_etDiag	:= GD.ET_Diag.Ok,
						i_etDiagExt	:= ET_DiagExt.Disabled,
						i_sMsg		:= '');
	END_IF
END_IF

DiagQuit();

CASE diState OF
	
	0:	(* Disable & exception state *)
	
	10:	(* Wait until diagnostics manager ready *)
		IF iq_stComStructure.i_xDiagnosticsManagerReady THEN
			
			SetDiagOutputs(	i_etDiag	:= GD.ET_Diag.Ok,
							i_etDiagExt	:= ET_DiagExt.WaitUntilDiagSourceRegistered,
							i_sMsg		:= '');
			diState := 20;
		END_IF

	20:	(* Wait until diag source registered *)	
		IF NOT iq_stComStructure.i_xDiagnosticsManagerReady THEN
			
			SetDiagOutputs(	i_etDiag	:= GD.ET_Diag.Ok,
							i_etDiagExt	:= ET_DiagExt.WaitUntilDiagnosticsManagerReady,
							i_sMsg		:= '');	
			diState := 10;
			RETURN;
	
		(* only write to register structure if no one else has done it in this cylce *)
		ELSIF (NOT iq_stComStructure.iq_stRegister.xUsed AND iq_stComStructure.iq_stRegister.udiNextId <> 0) THEN
			(* register *)
			iq_stComStructure.iq_stRegister.xUsed := TRUE;
			
			iq_stComStructure.iq_stRegister.sName		:= c_sName;
			iq_stComStructure.iq_stRegister.sTypeName	:= c_sTypeName;
			
			udiOwnSourceId := iq_stComStructure.iq_stRegister.udiNextId; (* register with this id; required for the following communication *)
		ELSE
			RETURN;
		END_IF
		
		q_xReady := TRUE;
		
		SetDiagOutputs(	i_etDiag	:= GD.ET_Diag.Ok,
						i_etDiagExt	:= ET_DiagExt.WaitForCommunication,
						i_sMsg		:= '');
		diState := 30;
	
	30:	(* Wait for communication *)	
		IF NOT iq_stComStructure.i_xDiagnosticsManagerReady THEN

			CancelWriting();
									
			udiOwnSourceId	:= 0;
			
			SetDiagOutputs(	i_etDiag	:= GD.ET_Diag.Ok,
							i_etDiagExt	:= ET_DiagExt.WaitUntilDiagnosticsManagerReady,
							i_sMsg		:= '');	
			diState := 10;
			RETURN;
			
		ELSIF (iq_stComStructure.i_udiComWithId = udiOwnSourceId) THEN		(* Am I adressed? *)
			
			WriteDiagDataControl();

		ELSE
			iq_stComStructure.q_lrProgress := 0.0;
			
			CancelWriting();
						
			SetDiagOutputs(	i_etDiag	:= GD.ET_Diag.Ok,
							i_etDiagExt	:= ET_DiagExt.WaitForCommunication,
							i_sMsg		:= '');
		END_IF
		
	100: (* Wait until disabled *)	
		IF NOT iq_stComStructure.i_xDiagnosticsManagerReady THEN

			CancelWriting();
									
			udiOwnSourceId	:= 0;
			
			SetDiagOutputs(	i_etDiag	:= GD.ET_Diag.Ok,
							i_etDiagExt	:= ET_DiagExt.Disabled,
							i_sMsg		:= '');	
	
		ELSIF (iq_stComStructure.i_udiComWithId = udiOwnSourceId) THEN		(* Am I adressed? *)
			
			WriteDiagDataControl();
			
		(* only write to register structure if no one else has done it in this cylce *)
		ELSIF (NOT iq_stComStructure.iq_stRegister.xUsed AND NOT iq_stComStructure.iq_stRegister.xUnsubscribe) AND 
			   NOT iq_stComStructure.i_xDiagnosticsActive THEN
			   
			iq_stComStructure.iq_stRegister.xUsed			:= TRUE;
			
			iq_stComStructure.iq_stRegister.xUnsubscribe	:= TRUE;
			iq_stComStructure.iq_stRegister.udiSourceId		:= udiOwnSourceId;
			
			q_xActive := FALSE;
			
			SetDiagOutputs(	i_etDiag	:= GD.ET_Diag.Ok,
							i_etDiagExt	:= ET_DiagExt.Disabled,
							i_sMsg		:= '');
		END_IF
END_CASE

IF q_xActive THEN	
	IF(diCmdExecState <> 0) THEN
		WriteDiagDataToFile();
		
		IF(iq_stComStructure.iq_diCmd <= 0) THEN
			diOldCmd := iq_stComStructure.iq_diCmd;
		END_IF
	END_IF	
END_IF

{attribute 'hide'}
METHOD CancelWriting : BOOL
VAR_INPUT
END_VAR
(* Deactivate writing if we are (for whatever reason) no longer adressed.
   May happen in case network connection with Diagnostics is disrupted or Source will be disabled *)

THIS^.diOldCmd			:= 0;
THIS^.diCmdExecState	:= 0;
END_METHOD

{attribute 'hide'}
METHOD DiagQuit : BOOL
VAR_INPUT
END_VAR
IF THIS^.i_xEnable AND THIS^.q_xActive AND THIS^.q_etDiag <> GD.ET_Diag.Ok AND THIS^.diState = 0 THEN

	THIS^.rtrigDiagQuit(CLK := THIS^.i_xDiagQuit);
	IF THIS^.rtrigDiagQuit.Q THEN
		CancelWriting();
									
		THIS^.udiOwnSourceId	:= 0;
		
		THIS^.fbTableWriter.FB_Init(bInitRetains := FALSE, bInCopyCode := FALSE);
			
		THIS^.q_xReady		:= TRUE;
		THIS^.q_etDiag		:= GD.ET_Diag.Ok;
		THIS^.q_etDiagExt	:= ET_DiagExt.WaitUntilDiagnosticsManagerReady;
		THIS^.q_sMsg		:= '';
	
		THIS^.diState := 10;
	END_IF

END_IF
END_METHOD

{attribute 'hide'}
METHOD ExceptionDuringWriting : BOOL
VAR_INPUT
END_VAR
(* exception during writing *)
CASE THIS^.etDiagExtTPL OF
	TPL.ET_DiagExt.HeaderStartAlreadySuccessfullyCalled,	// FB_TableWriter.HeaderStart	
	TPL.ET_DiagExt.FileIdNotSet,							// FB_TableWriter.HeaderStart							
	TPL.ET_DiagExt.FileIdInvalid,							// FB_TableWriter.HeaderStart & FB_TableWriter.HeaderAddColumn & FB_TableWriter.HeaderFinish & FB_TableWriter.RowStart & FB_TableWriter.RowValue & FB_TableWriter.TableEnd							
	TPL.ET_DiagExt.FileNotOpen,								// FB_TableWriter.HeaderStart & FB_TableWriter.HeaderAddColumn & FB_TableWriter.HeaderFinish & FB_TableWriter.RowStart & FB_TableWriter.RowValue & FB_TableWriter.TableEnd								
	TPL.ET_DiagExt.UnexpectedFeedback,						// FB_TableWriter.HeaderStart & FB_TableWriter.HeaderAddColumn & FB_TableWriter.HeaderFinish & FB_TableWriter.RowStart & FB_TableWriter.RowValue & FB_TableWriter.TableEnd								
	TPL.ET_DiagExt.HeaderStartNotCalled,					// FB_TableWriter.HeaderAddColumn								
	TPL.ET_DiagExt.HeaderStartNotSuccessfullyCalled,		// FB_TableWriter.HeaderAddColumn								
	TPL.ET_DiagExt.MaxNumberOfColumnsExceeded,				// FB_TableWriter.HeaderAddColumn						
	TPL.ET_DiagExt.NameInvalid,								// FB_TableWriter.HeaderAddColumn								
	TPL.ET_DiagExt.NoColumnsDefined,						// FB_TableWriter.HeaderFinish	
	TPL.ET_DiagExt.DefineHeaderFirst,						// FB_TableWriter.RowStart
	TPL.ET_DiagExt.RowStartedCallRowEndFirst,				// FB_TableWriter.RowStart
	TPL.ET_DiagExt.CallRowStartFirst,						// FB_TableWriter.RowValue
	TPL.ET_DiagExt.ColumnNumberRange,						// FB_TableWriter.RowValue
	TPL.ET_DiagExt.RowsStillOpen,							// FB_TableWriter.TableEnd
	TPL.ET_DiagExt.HeaderColumnIdInvalid:
	
		SetDiagOutputs(	i_etDiag	:= GD.ET_Diag.UnexpectedProgramBehavior,
						i_etDiagExt	:= ET_DiagExt.UnexpectedFeedback,
						i_sMsg		:= PDL.FC_MultiConcat(	i_sString1	:= 'FB_TableWriter: ', 
															i_sString2	:= GD.FC_EtDiagToString(THIS^.etDiag), 
															i_sString3	:= ' - ', 
															i_sString4	:= TPL.FC_EtDiagExtToString(THIS^.etDiagExtTPL), 
															q_etDiag	=> , 
															q_etDiagExt	=> )); 								
	ELSE
		SetDiagOutputs(	i_etDiag	:= GD.ET_Diag.UnexpectedProgramBehavior,
						i_etDiagExt	:= ET_DiagExt.UnexpectedFeedback,
						i_sMsg		:= PDL.FC_MultiConcat(	i_sString1	:= 'FB_TableWriter: ', 
															i_sString2	:= GD.FC_EtDiagToString(THIS^.etDiag), 
															i_sString3	:= ' - ', 
															i_sString4	:= TPL.FC_EtDiagExtToString(THIS^.etDiagExtTPL), 
															q_etDiag	=> , 
															q_etDiagExt	=> )); 						
END_CASE
		
CancelWriting();
END_METHOD

{attribute 'hide'}
METHOD SetDiagOutputs : BOOL
VAR_INPUT
	i_etDiag		: GD.ET_Diag;
	i_etDiagExt		: ET_DiagExt;
	i_sMsg			: STRING[80];
END_VAR
IF THIS^.q_etDiag = GD.ET_Diag.Ok OR i_etDiagExt = ET_DiagExt.Disabled THEN

	IF i_etDiag <> GD.ET_Diag.Ok OR i_etDiagExt = ET_DiagExt.Disabled THEN
		
		IF i_etDiag <> GD.ET_Diag.Ok THEN
			THIS^.iq_stComStructure.iq_diCmd := -THIS^.iq_stComStructure.iq_diCmd;
		END_IF
		
		IF i_etDiagExt = ET_DiagExt.Disabled THEN
			THIS^.q_xActive := FALSE;
			
			CancelWriting();
		END_IF
		
		THIS^.q_xReady := FALSE;
		THIS^.diState := 0;
	END_IF
	
	THIS^.q_etDiag		:= i_etDiag;
	THIS^.q_etDiagExt	:= i_etDiagExt;
	THIS^.q_sMsg		:= i_sMsg;

END_IF
END_METHOD

{attribute 'hide'}
METHOD WriteDiagDataControl : BOOL
VAR_INPUT
END_VAR
IF (THIS^.diOldCmd <> THIS^.iq_stComStructure.iq_diCmd AND THIS^.iq_stComStructure.iq_diCmd > 0) THEN
	
	THIS^.diOldCmd := THIS^.iq_stComStructure.iq_diCmd;
	
	(* new command, start execution *)
	CASE THIS^.iq_stComStructure.iq_diCmd OF
		
		1: (* write diag data to file *)
			IF (THIS^.iq_stComStructure.i_diFileId > 0) THEN
				
				SetDiagOutputs(	i_etDiag		:= GD.ET_Diag.Ok,
								i_etDiagExt		:= ET_DiagExt.WritingToFile,
								i_sMsg			:= '');
				
				THIS^.iq_stComStructure.q_lrProgress := 0.0;
				
				THIS^.fbTableWriter.diFileId := THIS^.iq_stComStructure.i_diFileId;
				
				THIS^.diCmdExecState := 1; (* start writing to file *)
			ELSE
				(* invalid file id *)
				SetDiagOutputs(	i_etDiag		:= GD.ET_Diag.InputParameterInvalid,
								i_etDiagExt		:= ET_DiagExt.FileIdInvalid,
								i_sMsg			:= CONCAT('Invalid file Id iq_stComStructure.i_diFileId: ', DINT_TO_STRING(THIS^.iq_stComStructure.i_diFileId)));
			END_IF
		ELSE
			(* unkown cmd *)
			SetDiagOutputs(	i_etDiag		:= GD.ET_Diag.InputParameterInvalid,
							i_etDiagExt		:= ET_DiagExt.CmdUnknown,
							i_sMsg			:= CONCAT('Unknown command iq_stComStructure.diCmd: ', DINT_TO_STRING(THIS^.iq_stComStructure.iq_diCmd)));

			CancelWriting();
	END_CASE
END_IF
END_METHOD

{attribute 'hide'}
METHOD WriteDiagDataToFile : BOOL
VAR_INPUT
END_VAR
TPL.FC_CanContinueWriting(iq_stCanContinueWriting := THIS^.iq_stComStructure.iq_stCanContinueWriting); (* loop as long as we can continue to write *)

WHILE (THIS^.iq_stComStructure.iq_stCanContinueWriting.xCanContinue) DO
	
	CASE THIS^.diCmdExecState OF
		1:
			(* start writing *)
			THIS^.fbTableWriter.HeaderStart(	i_sName					:= THIS^.c_sName, 
												i_sTypeName				:= THIS^.c_sTypeName, 
												i_sTitleEnglish			:= 'Example Data as Table', 
												i_sTitleGerman			:= 'Beispieldaten als Tabelle', 
												i_uiPrintRank			:= 14, 
												i_sEmptyListTextEnglish	:= 'No data available to show', 
												i_sEmptyListTextGerman	:= 'Keine Daten zum Anzeigen vorhanden',
												q_etDiag				=> THIS^.etDiag,
												q_etDiagExt				=> THIS^.etDiagExtTPL);
										
			IF THIS^.etDiag <> GD.ET_Diag.Ok THEN
				ExceptionDuringWriting();
				EXIT;
			END_IF
			
			THIS^.udiCName := THIS^.fbTableWriter.HeaderAddColumn(	i_sName			:= 'Name',
																	i_sTextEnglish	:= 'Name',
																	i_sTextGerman	:= 'Name',
																	i_uiWidth		:= 120,
																	q_etDiag		=> THIS^.etDiag,
																	q_etDiagExt		=> THIS^.etDiagExtTPL);
			IF THIS^.etDiag <> GD.ET_Diag.Ok THEN
				ExceptionDuringWriting();
				EXIT;
			END_IF

			THIS^.udiCValue := THIS^.fbTableWriter.HeaderAddColumn(	i_sName			:= 'Value',
																	i_sTextEnglish	:= 'Value',
																	i_sTextGerman	:= 'Wert',
																	i_uiWidth		:= 120,
																	q_etDiag		=> THIS^.etDiag,
																	q_etDiagExt		=> THIS^.etDiagExtTPL);
			IF THIS^.etDiag <> GD.ET_Diag.Ok THEN
				ExceptionDuringWriting();
				EXIT;
			END_IF

			THIS^.udiCC3 := THIS^.fbTableWriter.HeaderAddColumn(i_sName			:= 'Column3',
																i_sTextEnglish	:= 'Column3',
																i_sTextGerman	:= 'Spalte3',
																i_uiWidth		:= 120,
																q_etDiag		=> THIS^.etDiag,
																q_etDiagExt		=> THIS^.etDiagExtTPL);
			IF THIS^.etDiag <> GD.ET_Diag.Ok THEN
				ExceptionDuringWriting();
				EXIT;
			END_IF

			IF THIS^.udiCC3 <= 0 OR THIS^.udiCValue <= 0 OR THIS^.udiCName <= 0 THEN

				THIS^.etDiag		:= GD.ET_Diag.ExecutionAborted;
				THIS^.etDiagExtTPL	:= TPL.ET_DiagExt.HeaderColumnIdInvalid;

				ExceptionDuringWriting();
				EXIT;
			END_IF

			THIS^.fbTableWriter.HeaderFinish(	q_etDiag	=> THIS^.etDiag,
												q_etDiagExt	=> THIS^.etDiagExtTPL);
										
			IF THIS^.etDiag <> GD.ET_Diag.Ok THEN
				ExceptionDuringWriting();
				EXIT;
			END_IF

			THIS^.udiRowCounter := 1; (* start loop at index 1 *)

			THIS^.diCmdExecState := THIS^.diCmdExecState + 1;
			
		2:	(* loop over all rows *)

			IF (THIS^.udiRowCounter <= THIS^.c_udiMaxNumRows) THEN
				
				(* write row *)
				THIS^.fbTableWriter.RowStart(	q_etDiag	=> THIS^.etDiag,
												q_etDiagExt	=> THIS^.etDiagExtTPL);
										
				IF THIS^.etDiag <> GD.ET_Diag.Ok THEN
					ExceptionDuringWriting();
					EXIT;
				END_IF
				
				(* write values *)
				THIS^.fbTableWriter.RowValue(	i_udiColumnNumber	:= THIS^.udiCName, 
												i_sValue			:= CONCAT('name_',UDINT_TO_STRING(udiRowCounter)),
												q_etDiag			=> THIS^.etDiag,
												q_etDiagExt			=> THIS^.etDiagExtTPL);
										
				IF THIS^.etDiag <> GD.ET_Diag.Ok THEN
					ExceptionDuringWriting();
					EXIT;
				END_IF

				THIS^.fbTableWriter.RowValue(	i_udiColumnNumber	:= THIS^.udiCValue, 
												i_sValue			:= LREAL_TO_STRING((8000.0 - UDINT_TO_LREAL(udiRowCounter))/5),
												q_etDiag			=> THIS^.etDiag,
												q_etDiagExt			=> THIS^.etDiagExtTPL);
										
				IF THIS^.etDiag <> GD.ET_Diag.Ok THEN
					ExceptionDuringWriting();
					EXIT;
				END_IF

				THIS^.fbTableWriter.RowValue(	i_udiColumnNumber	:= THIS^.udiCC3, 
												i_sValue			:= UDINT_TO_STRING(udiRowCounter + 88),
												q_etDiag			=> THIS^.etDiag,
												q_etDiagExt			=> THIS^.etDiagExtTPL);
										
				IF THIS^.etDiag <> GD.ET_Diag.Ok THEN
					ExceptionDuringWriting();
					EXIT;
				END_IF
				
				THIS^.fbTableWriter.RowEnd(	q_etDiag	=> THIS^.etDiag,
											q_etDiagExt	=> THIS^.etDiagExtTPL);
										
				IF THIS^.etDiag <> GD.ET_Diag.Ok THEN
					ExceptionDuringWriting();
					EXIT;
				END_IF
			END_IF

			THIS^.iq_stComStructure.q_lrProgress := UDINT_TO_LREAL(THIS^.udiRowCounter) * LREAL#100.0 / MAX(UDINT_TO_LREAL(THIS^.c_udiMaxNumRows), LREAL#0.0001);

			THIS^.udiRowCounter := THIS^.udiRowCounter + 1;
			IF (THIS^.udiRowCounter > THIS^.c_udiMaxNumRows) THEN
				(* loop over all rows done *)
				THIS^.diCmdExecState := THIS^.diCmdExecState + 1;
			END_IF
		3:
			THIS^.fbTableWriter.TableEnd(	q_etDiag	=> THIS^.etDiag,
											q_etDiagExt	=> THIS^.etDiagExtTPL);
									
			IF THIS^.etDiag <> GD.ET_Diag.Ok THEN
				ExceptionDuringWriting();
				EXIT;
			END_IF
			
			(* done *)
			THIS^.iq_stComStructure.iq_diCmd := 0;

			SetDiagOutputs(	i_etDiag	:= GD.ET_Diag.Ok,
							i_etDiagExt	:= ET_DiagExt.DataSuccessfullyWritten,
							i_sMsg		:= '');					
	
			THIS^.diCmdExecState := 0;
			EXIT; (* exit the while loop *)
	END_CASE
	
	(* check again whether we can continue writing *)
	TPL.FC_CanContinueWriting(iq_stCanContinueWriting := THIS^.iq_stComStructure.iq_stCanContinueWriting);
END_WHILE
END_METHOD

END_FUNCTION_BLOCK

// LMC_PacDrive/Application/TemplateFullProgrammingFramework/Examples/ExampleDiagSources/FB_ExampleTreeDiagSource
FUNCTION_BLOCK FB_ExampleTreeDiagSource
VAR_INPUT
	i_xEnable			: BOOL;
	i_xDiagQuit			: BOOL;
END_VAR

VAR_IN_OUT
	iq_stComStructure	: TPL.ST_DiagnosticsManagerToDiagSource;
END_VAR

VAR_OUTPUT
	q_xActive			: BOOL;
	q_xReady			: BOOL;
	q_etDiag			: GD.ET_Diag := GD.ET_Diag.Ok;
	q_etDiagExt			: ET_DiagExt := ET_DiagExt.Disabled;
	q_sMsg				: STRING[80];
END_VAR

VAR
	xEnableFlag		: BOOL;
	diState			: DINT;
	
	udiOwnSourceId : UDINT := 0;
	
	fbTreeWriter	: TPL.FB_TreeWriter;

	diOldCmd	: DINT := 0;
	diCmdExecState : DINT := 0;

	uiMaxNodePerLevel : UINT := 7;

	uiLevelCounter : UINT := 1;
	auiNodeCounter : ARRAY[1..c_uiMaxLevel] OF UINT;
	uiNodeId : UINT := 1;
	lrSumNodes : LREAL := 1;

	uiTmp : UINT := 0;
	
	etDiag			: GD.ET_Diag;
	etDiagExtTPL	: TPL.ET_DiagExt;
	sMsg			: STRING[80];
	
	rtrigDiagQuit	: Standard.R_TRIG;
END_VAR

VAR CONSTANT
	c_sName : STRING[TPL.Gc_udiTableWriterMaxNameLength] := 'I_am_a_Tree';
	c_sTypeName : STRING[TPL.Gc_udiTableWriterMaxNameLength] := 'ExampleTreeDiagSource';
	c_uiMaxLevel : UINT := 5;
END_VAR

IF i_xEnable AND NOT xEnableFlag THEN
	xEnableFlag := TRUE;
	
	q_xActive := TRUE;
	
	SetDiagOutputs(	i_etDiag	:= GD.ET_Diag.Ok,
					i_etDiagExt	:= ET_DiagExt.WaitUntilDiagnosticsManagerReady,
					i_sMsg		:= '');	
	diState := 10;
	
ELSIF NOT i_xEnable AND xEnableFlag THEN
	xEnableFlag := FALSE;
		
	IF udiOwnSourceId <> 0 THEN		
		SetDiagOutputs(	i_etDiag	:= GD.ET_Diag.Ok,
						i_etDiagExt	:= ET_DiagExt.WaitUntilDisabled,
						i_sMsg		:= '');
		diState := 100;
		
	ELSIF udiOwnSourceId = 0 THEN		
		SetDiagOutputs(	i_etDiag	:= GD.ET_Diag.Ok,
						i_etDiagExt	:= ET_DiagExt.Disabled,
						i_sMsg		:= '');
	END_IF
END_IF

DiagQuit();

CASE diState OF
	
	0:	(* Disable & exception state *)
	
	10:	(* Wait until diagnostics manager ready *)
		IF iq_stComStructure.i_xDiagnosticsManagerReady THEN
			
			SetDiagOutputs(	i_etDiag	:= GD.ET_Diag.Ok,
							i_etDiagExt	:= ET_DiagExt.WaitUntilDiagSourceRegistered,
							i_sMsg		:= '');
			diState := 20;
		END_IF

	20:	(* Wait until diag source registered *)	
		IF NOT iq_stComStructure.i_xDiagnosticsManagerReady THEN
			
			SetDiagOutputs(	i_etDiag	:= GD.ET_Diag.Ok,
							i_etDiagExt	:= ET_DiagExt.WaitUntilDiagnosticsManagerReady,
							i_sMsg		:= '');	
			diState := 10;
			RETURN;
	
		(* only write to register structure if no one else has done it in this cylce *)
		ELSIF (NOT iq_stComStructure.iq_stRegister.xUsed AND iq_stComStructure.iq_stRegister.udiNextId <> 0) THEN
			(* register *)
			iq_stComStructure.iq_stRegister.xUsed := TRUE;
			
			iq_stComStructure.iq_stRegister.sName		:= c_sName;
			iq_stComStructure.iq_stRegister.sTypeName	:= c_sTypeName;
			
			udiOwnSourceId := iq_stComStructure.iq_stRegister.udiNextId; (* register with this id; required for the following communication *)
		ELSE
			RETURN;
		END_IF
		
		q_xReady := TRUE;
		
		SetDiagOutputs(	i_etDiag	:= GD.ET_Diag.Ok,
						i_etDiagExt	:= ET_DiagExt.WaitForCommunication,
						i_sMsg		:= '');
		diState := 30;
	
	30:	(* Wait for communication *)	
		IF NOT iq_stComStructure.i_xDiagnosticsManagerReady THEN

			CancelWriting();
									
			udiOwnSourceId	:= 0;
			
			SetDiagOutputs(	i_etDiag	:= GD.ET_Diag.Ok,
							i_etDiagExt	:= ET_DiagExt.WaitUntilDiagnosticsManagerReady,
							i_sMsg		:= '');	
			diState := 10;
			RETURN;
			
		ELSIF (iq_stComStructure.i_udiComWithId = udiOwnSourceId) THEN		(* Am I adressed? *)
			
			WriteDiagDataControl();

		ELSE
			iq_stComStructure.q_lrProgress := 0.0;
			
			CancelWriting();
						
			SetDiagOutputs(	i_etDiag	:= GD.ET_Diag.Ok,
							i_etDiagExt	:= ET_DiagExt.WaitForCommunication,
							i_sMsg		:= '');
		END_IF
		
	100: (* Wait until disabled *)	
		IF NOT iq_stComStructure.i_xDiagnosticsManagerReady THEN

			CancelWriting();
									
			udiOwnSourceId	:= 0;
			
			SetDiagOutputs(	i_etDiag	:= GD.ET_Diag.Ok,
							i_etDiagExt	:= ET_DiagExt.Disabled,
							i_sMsg		:= '');	
	
		ELSIF (iq_stComStructure.i_udiComWithId = udiOwnSourceId) THEN		(* Am I adressed? *)
			
			WriteDiagDataControl();
			
		(* only write to register structure if no one else has done it in this cylce *)
		ELSIF (NOT iq_stComStructure.iq_stRegister.xUsed AND NOT iq_stComStructure.iq_stRegister.xUnsubscribe) AND 
			   NOT iq_stComStructure.i_xDiagnosticsActive THEN
			   
			iq_stComStructure.iq_stRegister.xUsed			:= TRUE;
			
			iq_stComStructure.iq_stRegister.xUnsubscribe	:= TRUE;
			iq_stComStructure.iq_stRegister.udiSourceId		:= udiOwnSourceId;
			
			q_xActive := FALSE;
			
			SetDiagOutputs(	i_etDiag	:= GD.ET_Diag.Ok,
							i_etDiagExt	:= ET_DiagExt.Disabled,
							i_sMsg		:= '');
		END_IF
END_CASE

IF q_xActive THEN	
	IF(diCmdExecState <> 0) THEN
		WriteDiagDataToFile();
		
		IF(iq_stComStructure.iq_diCmd <= 0) THEN
			diOldCmd := iq_stComStructure.iq_diCmd;
		END_IF
	END_IF	
END_IF

{attribute 'hide'}
METHOD CancelWriting : BOOL
VAR_INPUT
END_VAR
(* Deactivate writing if we are (for whatever reason) no longer adressed.
   May happen in case network connection with Diagnostics is disrupted or Source will be disabled *)

THIS^.diOldCmd			:= 0;
THIS^.diCmdExecState	:= 0;
END_METHOD

{attribute 'hide'}
METHOD DiagQuit : BOOL
VAR_INPUT
END_VAR
IF THIS^.i_xEnable AND THIS^.q_xActive AND THIS^.q_etDiag <> GD.ET_Diag.Ok AND THIS^.diState = 0 THEN

	THIS^.rtrigDiagQuit(CLK := THIS^.i_xDiagQuit);
	IF THIS^.rtrigDiagQuit.Q THEN
		CancelWriting();
									
		THIS^.udiOwnSourceId	:= 0;
		
		THIS^.fbTreeWriter.FB_Init(bInitRetains := FALSE, bInCopyCode := FALSE);
			
		THIS^.q_xReady		:= TRUE;
		THIS^.q_etDiag		:= GD.ET_Diag.Ok;
		THIS^.q_etDiagExt	:= ET_DiagExt.WaitUntilDiagnosticsManagerReady;
		THIS^.q_sMsg		:= '';
	
		THIS^.diState := 10;
	END_IF

END_IF
END_METHOD

{attribute 'hide'}
METHOD ExceptionDuringWriting : BOOL
VAR_INPUT
END_VAR
(* exception during writing *)
CASE THIS^.etDiagExtTPL OF
	TPL.ET_DiagExt.TreeStartAlreadySuccessfullyCalled,		// FB_TreeWriter.TreeStart	
	TPL.ET_DiagExt.FileIdNotSet,							// FB_TreeWriter.TreeStart							
	TPL.ET_DiagExt.FileIdInvalid,							// FB_TreeWriter.TreeStart & FB_TreeWriter.NodeStart & FB_TreeWriter.Parameter & FB_TreeWriter.NodeEnd & FB_TreeWriter.TreeEnd								
	TPL.ET_DiagExt.FileNotOpen,								// FB_TreeWriter.TreeStart & FB_TreeWriter.NodeStart & FB_TreeWriter.Parameter & FB_TreeWriter.NodeEnd & FB_TreeWriter.TreeEnd								
	TPL.ET_DiagExt.UnexpectedFeedback,						// FB_TreeWriter.TreeStart & FB_TreeWriter.NodeStart & FB_TreeWriter.Parameter & FB_TreeWriter.NodeEnd & FB_TreeWriter.TreeEnd								
	TPL.ET_DiagExt.TreeStartNotCalled,						// FB_TreeWriter.NodeStart								
	TPL.ET_DiagExt.TreeStartNotSuccessfullyCalled,			// FB_TreeWriter.NodeStart								
	TPL.ET_DiagExt.NoMoreNodeOpen,							// FB_TreeWriter.Parameter & FB_TreeWriter.NodeEnd						
	TPL.ET_DiagExt.CallTreeStartFirst,						// FB_TreeWriter.TreeEnd								
	TPL.ET_DiagExt.NodesStillOpen:							// FB_TreeWriter.TreeEnd	
	
		SetDiagOutputs(	i_etDiag	:= GD.ET_Diag.UnexpectedProgramBehavior,
						i_etDiagExt	:= ET_DiagExt.UnexpectedFeedback,
						i_sMsg		:= PDL.FC_MultiConcat(	i_sString1	:= 'FB_TreeWriter: ', 
															i_sString2	:= GD.FC_EtDiagToString(THIS^.etDiag), 
															i_sString3	:= ' - ', 
															i_sString4	:= TPL.FC_EtDiagExtToString(THIS^.etDiagExtTPL), 
															q_etDiag	=> , 
															q_etDiagExt	=> )); 								
	ELSE
		SetDiagOutputs(	i_etDiag	:= GD.ET_Diag.UnexpectedProgramBehavior,
						i_etDiagExt	:= ET_DiagExt.UnexpectedFeedback,
						i_sMsg		:= PDL.FC_MultiConcat(	i_sString1	:= 'FB_TreeWriter: ', 
															i_sString2	:= GD.FC_EtDiagToString(THIS^.etDiag), 
															i_sString3	:= ' - ', 
															i_sString4	:= TPL.FC_EtDiagExtToString(THIS^.etDiagExtTPL), 
															q_etDiag	=> , 
															q_etDiagExt	=> )); 						
END_CASE
		
CancelWriting();
END_METHOD

{attribute 'hide'}
METHOD SetDiagOutputs : BOOL
VAR_INPUT
	i_etDiag		: GD.ET_Diag;
	i_etDiagExt		: ET_DiagExt;
	i_sMsg			: STRING[80];
END_VAR
IF THIS^.q_etDiag = GD.ET_Diag.Ok OR i_etDiagExt = ET_DiagExt.Disabled THEN

	IF i_etDiag <> GD.ET_Diag.Ok OR i_etDiagExt = ET_DiagExt.Disabled THEN
		
		IF i_etDiag <> GD.ET_Diag.Ok THEN
			THIS^.iq_stComStructure.iq_diCmd := -THIS^.iq_stComStructure.iq_diCmd;
		END_IF
		
		IF i_etDiagExt = ET_DiagExt.Disabled THEN
			THIS^.q_xActive := FALSE;
			
			CancelWriting();
		END_IF
		
		THIS^.q_xReady := FALSE;
		THIS^.diState := 0;
	END_IF
	
	THIS^.q_etDiag		:= i_etDiag;
	THIS^.q_etDiagExt	:= i_etDiagExt;
	THIS^.q_sMsg		:= i_sMsg;

END_IF
END_METHOD

{attribute 'hide'}
METHOD WriteDiagDataControl : BOOL
VAR_INPUT
END_VAR
IF (THIS^.diOldCmd <> THIS^.iq_stComStructure.iq_diCmd AND THIS^.iq_stComStructure.iq_diCmd > 0) THEN
	
	THIS^.diOldCmd := THIS^.iq_stComStructure.iq_diCmd;
	
	(* new command, start execution *)
	CASE THIS^.iq_stComStructure.iq_diCmd OF
		
		1: (* write diag data to file *)
			IF (THIS^.iq_stComStructure.i_diFileId > 0) THEN
				
				SetDiagOutputs(	i_etDiag		:= GD.ET_Diag.Ok,
								i_etDiagExt		:= ET_DiagExt.WritingToFile,
								i_sMsg			:= '');
				
				THIS^.iq_stComStructure.q_lrProgress := 0.0;
				
				THIS^.fbTreeWriter.diFileId := THIS^.iq_stComStructure.i_diFileId;
				
				THIS^.diCmdExecState := 1; (* start writing to file *)
			ELSE
				(* invalid file id *)
				SetDiagOutputs(	i_etDiag		:= GD.ET_Diag.InputParameterInvalid,
								i_etDiagExt		:= ET_DiagExt.FileIdInvalid,
								i_sMsg			:= CONCAT('Invalid file Id iq_stComStructure.i_diFileId: ', DINT_TO_STRING(THIS^.iq_stComStructure.i_diFileId)));
			END_IF
		ELSE
			(* unkown cmd *)
			SetDiagOutputs(	i_etDiag		:= GD.ET_Diag.InputParameterInvalid,
							i_etDiagExt		:= ET_DiagExt.CmdUnknown,
							i_sMsg			:= CONCAT('Unknown command iq_stComStructure.diCmd: ', DINT_TO_STRING(THIS^.iq_stComStructure.iq_diCmd)));

			CancelWriting();
	END_CASE
END_IF
END_METHOD

{attribute 'hide'}
METHOD WriteDiagDataToFile : BOOL
VAR_INPUT
END_VAR
TPL.FC_CanContinueWriting(iq_stCanContinueWriting := THIS^.iq_stComStructure.iq_stCanContinueWriting); (* loop as long as we can continue to write *)

WHILE (THIS^.iq_stComStructure.iq_stCanContinueWriting.xCanContinue) DO
	
	CASE THIS^.diCmdExecState OF
		1:
			(* start writing *)
			THIS^.fbTreeWriter.TreeStart(	i_sName					:= THIS^.c_sName, 
											i_sTypeName				:= THIS^.c_sTypeName, 
											i_sTitleEnglish			:= 'Example data as tree', 
											i_sTitleGerman			:= 'Beispieldaten als Baum', 
											i_uiPrintRank			:= 14, 
											i_sEmptyListTextEnglish	:= 'No data available to show', 
											i_sEmptyListTextGerman	:= 'Keine Daten zum Anzeigen vorhanden',
											q_etDiag				=> THIS^.etDiag,
											q_etDiagExt				=> THIS^.etDiagExtTPL);
									
			IF THIS^.etDiag <> GD.ET_Diag.Ok THEN
				ExceptionDuringWriting();
				EXIT;
			END_IF

			FOR THIS^.uiLevelCounter := 1 TO THIS^.c_uiMaxLevel DO
				THIS^.auiNodeCounter[uiLevelCounter] := 1;
			END_FOR

			THIS^.uiNodeId := 1;

			THIS^.lrSumNodes := ((1 - EXPT(THIS^.uiMaxNodePerLevel, THIS^.c_uiMaxLevel + 1)) / (1 - THIS^.uiMaxNodePerLevel));

			THIS^.uiLevelCounter := 1; (* start loop at index 1 *)

			THIS^.diCmdExecState := THIS^.diCmdExecState + 1;
		2:
			IF (THIS^.auiNodeCounter[THIS^.uiLevelCounter] <= THIS^.uiMaxNodePerLevel) THEN
				(* don't need to go up again, can create more nodes on this level *)

				(* create another subnode and go down *)
				(* create another node *)
				THIS^.uiNodeId := 0;
				THIS^.auiNodeCounter[THIS^.uiLevelCounter] := THIS^.auiNodeCounter[THIS^.uiLevelCounter] + 1;
				
				FOR THIS^.uiTmp := 1 TO THIS^.uiLevelCounter DO
					THIS^.uiNodeId := THIS^.uiNodeId * 100 + (THIS^.auiNodeCounter[THIS^.uiTmp] - 1);
				END_FOR
				
				THIS^.fbTreeWriter.NodeStart(	i_sName		:= CONCAT('Knoten_', UINT_TO_STRING(uiNodeId)),
												q_etDiag	=> THIS^.etDiag,
												q_etDiagExt	=> THIS^.etDiagExtTPL);
										
				IF THIS^.etDiag <> GD.ET_Diag.Ok THEN
					ExceptionDuringWriting();
					EXIT;
				END_IF
				
					THIS^.fbTreeWriter.Parameter(	i_sName		:= 'something', 
													i_sValue	:= LREAL_TO_STRING(UINT_TO_LREAL(uiLevelCounter * auiNodeCounter[uiLevelCounter]) / UINT_TO_LREAL(uiNodeId)),
													q_etDiag	=> THIS^.etDiag,
													q_etDiagExt	=> THIS^.etDiagExtTPL);
											
					IF THIS^.etDiag <> GD.ET_Diag.Ok THEN
						ExceptionDuringWriting();
						EXIT;
					END_IF

				THIS^.uiLevelCounter := THIS^.uiLevelCounter + 1;

				IF (THIS^.uiLevelCounter > THIS^.c_uiMaxLevel) THEN
					(* go up again *)
					THIS^.fbTreeWriter.NodeEnd(	q_etDiag	=> THIS^.etDiag,
												q_etDiagExt	=> THIS^.etDiagExtTPL);	
											
					IF THIS^.etDiag <> GD.ET_Diag.Ok THEN
						ExceptionDuringWriting();
						EXIT;
					END_IF

					THIS^.uiLevelCounter := THIS^.uiLevelCounter - 1;
				END_IF
			ELSE
				(* go up again *)
				THIS^.fbTreeWriter.NodeEnd(	q_etDiag	=> THIS^.etDiag,
											q_etDiagExt	=> THIS^.etDiagExtTPL);	
										
				IF THIS^.etDiag <> GD.ET_Diag.Ok THEN
					ExceptionDuringWriting();
					EXIT;
				END_IF

				THIS^.auiNodeCounter[THIS^.uiLevelCounter] := 1; (* reset node counter of level *)

				THIS^.uiLevelCounter := THIS^.uiLevelCounter - 1;
				IF (THIS^.uiLevelCounter <= 1) THEN
					(* loop over all nodes and levels done *)
					THIS^.diCmdExecState := THIS^.diCmdExecState + 1;
				END_IF
			END_IF

			THIS^.iq_stComStructure.q_lrProgress := UINT_TO_LREAL(THIS^.auiNodeCounter[1]) * LREAL#100.0 / MAX(THIS^.lrSumNodes,0.0001);

		3:
			THIS^.fbTreeWriter.TreeEnd(	q_etDiag	=> THIS^.etDiag,
										q_etDiagExt	=> THIS^.etDiagExtTPL);	
									
			IF THIS^.etDiag <> GD.ET_Diag.Ok THEN
				ExceptionDuringWriting();
				EXIT;
			END_IF
			(* done *)
			
			(* signal command execution *)
			THIS^.iq_stComStructure.iq_diCmd := 0;
			
			SetDiagOutputs(	i_etDiag	:= GD.ET_Diag.Ok,
							i_etDiagExt	:= ET_DiagExt.DataSuccessfullyWritten,
							i_sMsg		:= '');		
			
			THIS^.diCmdExecState := 0;
			EXIT; (* exit the while loop *)
	END_CASE
	
	(* check again whether we can continue writing *)
	TPL.FC_CanContinueWriting(iq_stCanContinueWriting := THIS^.iq_stComStructure.iq_stCanContinueWriting);
END_WHILE
END_METHOD

END_FUNCTION_BLOCK

// LMC_PacDrive/Application/TemplateFullProgrammingFramework/TaskCalls/SR_Logging
PROGRAM SR_Logging
VAR
	fbLogDataControl	: TPL.FB_LogDataControl;
END_VAR

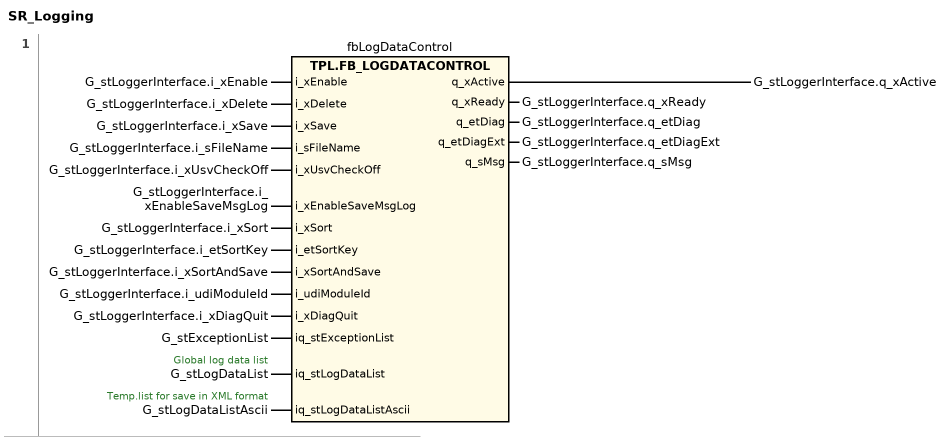
// NETWORK 1
//   G_stLogDataList: Global log data list
//   G_stLogDataListAscii: Temp.list for save in XML format
fbLogDataControl(
    i_xEnable := G_stLoggerInterface.i_xEnable,
    i_xDelete := G_stLoggerInterface.i_xDelete,
    i_xSave := G_stLoggerInterface.i_xSave,
    i_sFileName := G_stLoggerInterface.i_sFileName,
    i_xUsvCheckOff := G_stLoggerInterface.i_xUsvCheckOff,
    i_xEnableSaveMsgLog := G_stLoggerInterface.i_xEnableSaveMsgLog,
    i_xSort := G_stLoggerInterface.i_xSort,
    i_etSortKey := G_stLoggerInterface.i_etSortKey,
    i_xSortAndSave := G_stLoggerInterface.i_xSortAndSave,
    i_udiModuleId := G_stLoggerInterface.i_udiModuleId,
    i_xDiagQuit := G_stLoggerInterface.i_xDiagQuit,
    iq_stExceptionList := G_stExceptionList,
    iq_stLogDataList := G_stLogDataList,
    iq_stLogDataListAscii := G_stLogDataListAscii,
    q_xReady => G_stLoggerInterface.q_xReady,
    q_etDiag => G_stLoggerInterface.q_etDiag,
    q_etDiagExt => G_stLoggerInterface.q_etDiagExt,
    q_sMsg => G_stLoggerInterface.q_sMsg); // TPL.FB_LOGDATACONTROL
G_stLoggerInterface.q_xActive := fbLogDataControl.q_xActive;

END_PROGRAM

// LMC_PacDrive/Application/TemplateFullProgrammingFramework/TaskCalls/SR_HWCopyIO
PROGRAM SR_HWCopyIO

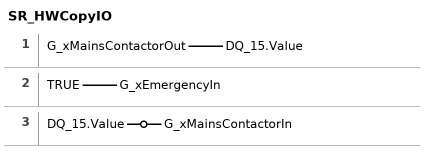
// NETWORK 1
DQ_15.Value := G_xMainsContactorOut;

// NETWORK 2
G_xEmergencyIn := TRUE;

// NETWORK 3
G_xMainsContactorIn := NOT DQ_15.Value;

END_PROGRAM

// LMC_PacDrive/Application/TemplateFullProgrammingFramework/TaskCalls/SR_VisControl
PROGRAM SR_VisControl
VAR CONSTANT
	c_udiMaxHierarchyLevels	: UDINT := 10;
	c_stEmptyCmdTableStep	: TPL.ST_Cmd := (	sTitle			:= '',
												diStep			:= 0,
												udiModuleName	:= 0,
												diCmd			:= 0,
												timTimeOut		:= T#60S,
												xEndCmd			:= FALSE);
END_VAR
VAR (*User specific variables*)
	
END_VAR
VAR
	iState							: INT:= 0;
	vpq_xDoEnable 					: BOOL:= FALSE;
	xEnableFlag 					: BOOL;
	iDoEnableCycleCounter			: INT:=0;
	
	IFB_RTOPMode					: STANDARD.R_TRIG;

(* Cmd table of main machine on VIS_Main *)
	pstStep 						: POINTER TO TPL.ST_Cmd;
	udiCounter						: UDINT;
	
	vpq_astActualCmdTableMain	: ARRAY [1..10] OF TPL.ST_Cmd;
	vpq_udiNumberOfCmdStepsMain	: UDINT;
	vpq_sCmdTitelMain		: STRING;
	vpiq_udiIndexMinMain		: UDINT := 1;
	udiIndexMaxMainTable			: UDINT := 1;
	udiIndexOldMainTable			: UDINT := 1;
	
	vpq_xDisableScrollUpMain	: BOOL;
	vpq_xDisableScrollDownMain	: BOOL;

	(* Visualization of the main machine on the VIS_Main *)
	vpq_stMachineInterface				: TPL.ST_StandardModuleInterface;
	
	vpq_xMachineInException				: BOOL;	
	vpq_etMainModuleControllerDiag		: GD.ET_Diag;
	vpq_etMainModuleControllerDiagExt	: TPL.ET_DiagExt;
	vpq_sMainModuleControllerMsg			: STRING[80];

(*Exception*)
	vpiq_xTestUserException1				: BOOL;
	xTestUserException1Old					: BOOL;
	vpiq_xTestUserException2				: BOOL;
	xTestUserException2Old					: BOOL;
	vpiq_xTestUserException3				: BOOL;
	xTestUserException3Old					: BOOL;
	vpiq_xTestUserException4				: BOOL;
	xTestUserException4Old					: BOOL;
	vpiq_xTestUserException5				: BOOL;
	xTestUserException5Old					: BOOL;

	vpq_udiReactionIndexMin				: UDINT := 1;
	udiReactionIndexMax				: UDINT := 1;
	udiReactionIndexOld				: UDINT := 1;
	vpq_axReaction						: ARRAY[1..10] OF BOOL;
	
	udiCount						: UDINT;
	stActiveReactions				: TPL.ST_Reaction;
	vpiq_xReactionUp						: BOOL;
	vpiq_xReactionDown					: BOOL;

(*Vis*)
	vpiq_xShowControlFrame			: BOOL;
	vpiq_xShowModuleInterface		: BOOL;
	vpiq_iPositionX					: INT;
	vpiq_iPositionY					: INT;

	vpq_xShowLogDataListDetails				: BOOL := FALSE;
	vpiq_xButtonLogDataListDetails			: BOOL := FALSE;

	(* Visualization of the actCmdTable of the current module *)
	pstEQCMDTable							: POINTER TO TPL.ST_Cmd;		(* Pointer to active CMD Table *)
	pstEQCMDTableEntry						: POINTER TO TPL.ST_Cmd;
	vpq_astActualCmdTableModule				: ARRAY[1..10] OF TPL.ST_Cmd;
	vpiq_udiIndexMinModule						: UDINT := 1;
	udiEQTableIndexMax						: UDINT := 1;
	udiEQTableIndexOld						: UDINT := 1;
	vpq_udiNumberOfCmdStepsModule			: UDINT := 0;
	pstEQCMDTableListEntry					: POINTER TO TPL.ST_CmdTable;
	vpq_sCmdTitleModule						: STRING[80];
	udiEQTableStepCountOld					: UDINT;

	(* Navigation in the command table *)
	vpq_xDisableScrollUpModule				: BOOL;
	vpq_xDisableScrollDownModule			: BOOL;
	vpq_xDisplayCmdTable					: BOOL;

	(* 2d navigation buttons *)
	vpiq_xNavUp								: BOOL;
	vpiq_xNavDown							: BOOL;
	vpiq_xNavLeft							: BOOL;
	vpiq_xNavRight							: BOOL;
	vpq_xEnableNavUp						: BOOL;
	vpq_xEnableNavDown						: BOOL;
	vpq_xEnableNavLeft						: BOOL;
	vpq_xEnableNavRight						: BOOL;
	vpq_sNameNavUp							: STRING[80];
	vpq_sNameNavDown						: STRING[80];
	vpq_sNameNavLeft						: STRING[80];
	vpq_sNameNavRight						: STRING[80];

	(* Navigation flags *)
	pstCurrentParent						: POINTER TO TPL.ST_StandardModuleInterface;
	pstCurrent								: POINTER TO TPL.ST_StandardModuleInterface;
	xCurrentIsNoNodeModule    				: BOOL;
	dwCurrentAddInterface					: DWORD;
	xUpdateForOtherFBs						: BOOL;
	audiHierarchy							: ARRAY[1..c_udiMaxHierarchyLevels] OF UDINT; (* Selected modules in each level of the hierarchy *)
	udiCurrentLevel							: UDINT := 1; (* Level of the hierarchy we are working on*)
	udiCurrentLevelSize						: UDINT := 1;
	xCurrentHasSubModules					: BOOL := FALSE;
	pstTmp									: POINTER TO TPL.ST_StandardModuleInterface;
	pdwTmp									: POINTER TO DWORD;

	xUpdateData 							: BOOL := FALSE;
	dwDummy									: DWORD;

	vpq_xButtonSetJogTargetInvisible		: BOOL := FALSE;
	vpiq_xButtonSetCurrentAsJogTarget					: BOOL;
	vpq_xCurrentIsJogTarget						: BOOL := FALSE;
	udiSetAsJogTarget						: UDINT;
//	udiSetAsJogTargetNum					: UDINT;
	IFB_FTrigxCurrentIsJogTarget			: STANDARD.F_TRIG;

	(* Direct navigation buttons *)
	axClearBoolA5							: ARRAY[1..5] OF BOOL;
	
	vpiq_xModuleListDown							: BOOL; (* Module table scroll buttons *)
	vpq_xDisableModuleListDown					: BOOL;
	vpiq_xModuleListUp							: BOOL;
	vpq_xDisableModuleListUp						: BOOL;
	vpiq_axModuleList							: ARRAY[1..5] OF BOOL;
	vpiq_axControlModuleList						: ARRAY[1..5] OF BOOL;
	vpq_axDisableModuleList						: ARRAY[1..5] OF BOOL;
	vpq_axActiveModuleList						: ARRAY[1..5] OF BOOL; (* Highlight active module *)
	vpq_axControlModuleActive						: ARRAY[1..5] OF BOOL; (* Highlight active control module *)
	vpq_audiIdModuleList							: ARRAY[1..5] OF UDINT; (* Module ids *)
	vpq_axIdModuleListValid					: ARRAY[1..5] OF BOOL;
	vpq_axControlModuleValid					: ARRAY[1..5] OF BOOL;
	audiControlModuleNumber					: ARRAY[1..5] OF UDINT;
	vpq_asNameModuleList						: ARRAY[1..5] OF STRING[80]; (* Module name *)
	vpq_asToolTipControlModuleList				: ARRAY[1..5] OF STRING[80];
	vpq_asControlModuleButtonName				: ARRAY[1..5] OF STRING[60];
	udiNumberOfControlModulesLevel2			: UDINT;

	vpiq_xSubModuleListDown					: BOOL;
	vpq_xDisableSubModuleListDown			: BOOL;
	vpiq_xSubModuleListUp					: BOOL;
	vpq_xDisableSubModuleListUp				: BOOL;
	
	vpiq_axSubModuleList							: ARRAY[1..5] OF BOOL;
	vpq_axDisableSubModuleList					: ARRAY[1..5] OF BOOL;
	vpq_axActiveSubModuleList					: ARRAY[1..5] OF BOOL; (* Highlight active module *)
	vpq_audiIdSubModuleList					: ARRAY[1..5] OF UDINT; (* Module ids *)
	vpq_axIdSubModuleListValid						: ARRAY[1..5] OF BOOL;
	vpq_asNameSubModuleList						: ARRAY[1..5] OF STRING[60]; (* Module names *)
	vpiq_axSubControlModuleList					: ARRAY[1..5] OF BOOL;
	vpq_axSubControlModuleValid					: ARRAY[1..5] OF BOOL;
	audiSubControlModuleID					: ARRAY[1..5] OF UDINT;
	vpq_asToolTipSubControlModuleList			: ARRAY[1..5] OF STRING[80];
	vpq_axSubControlModuleActive					: ARRAY[1..5] OF BOOL;
	vpq_asSubControlModuleButtonName			: ARRAY[1..5] OF STRING[60];
	udiCurrentLevel3Size					: UDINT := 0; (* How many submodules does the current module have on level 2 *)
	pstCurrentFirstLevel3Module				: POINTER TO TPL.ST_StandardModuleInterface;
	udiCurrentNumberOfControlModules 		: UDINT;

	(*Variables for selecting control modules *)
	vpq_udiActiveControlModuleNumber				: UDINT;
	pstCurrentNodeInterface						: POINTER TO TPL.ST_StandardModuleInterface;
	pstControlModuleInterface					: POINTER TO TPL.ST_ControlModuleInterface;
	pstCurrentControlModuleStandardInterface	: POINTER TO TPL.ST_ControlModuleInterface;
	pstTempCtrlModule							: POINTER TO TPL.ST_ControlModuleInterface;
	stCurrentControlModuleStandardInterface		: TPL.ST_ControlModuleInterface;
	udiControlModuleSelectedInLevel				: UDINT;
	xControlModuleSelected						: BOOL;
	xCurrentHasControlModules					: BOOL;
	pstCurrentLevel2							: POINTER TO TPL.ST_StandardModuleInterface;

	(* Direct navigation flags *)
	udiMinModuleList						: UDINT;
	udiMinSubModuleList						: UDINT;

	(* Struct for displaying values of the current module *)
	vpq_stCurrentModuleStandardInterface		: TPL.ST_StandardModuleInterface;
	vpq_sCurrentModuleReaction				: STRING[255];
	stDummyStandardInterface				: TPL.ST_StandardModuleInterface;
	
	(* Exceptions the vis can create *)
	stPointerException						: TPL.ST_Exception;
	xPointerExceptionActive					: BOOL;


	udiSetAsCurrentModule					: UDINT; (* If <> 0, specifies the ID of a module, to set as current module *)

	(* Flags of the SetCurrentModule action *)
	udiTmp2									: UDINT;
	udiTmp									: UDINT;


	(* Inputs, for module control *)
	vpiq_diCmdToSet								: DINT;
	vpiq_diStartStepToSet					: DINT;
	vpiq_xSetCmdClicked							: BOOL; (* Set by the vis, reset by SR_VisControl, if true, diCmdToSet is written to the CMD of the current module *)
	xDiagQuit_Touch						: BOOL; (* Set by the vis, if true, the DiagQuit Input of the module is set *)
	xDiagQuit_WasTouched					: BOOL;	(* Internal flag *)
	vpiq_xEnableModuleClicked					: BOOL; (* Set by the vis, reset by SR_VisControl, if true, the xEnable of the module is toggled *)

	stModuleReactions						: TPL.ST_Reaction;
	vpiq_xModuleReactionUp						: BOOL;
	vpiq_xModuleReactionDown						: BOOL;
	vpq_udiModuleReactionIndexMin				: UDINT := 1;
	udiModuleReactionIndexMax				: UDINT := 1;
	udiModuleReactionIndexOld				: UDINT := 1;
	vpq_axModuleReaction						: ARRAY[1..10] OF BOOL;
	udiCount2								: UDINT;
	udiMaxValue								: UDINT;


	(*FR_ExceptionList, navigation in the global ExceptionList*)
	vpiq_udiExceptionListIndexMin			: UDINT := 1;
	vpq_asReaction							: ARRAY[1..10] OF STRING[80];
	vpq_udiExceptionListIndexMax				: UDINT := 1;
	vpq_xDisplayScrollDown					: BOOL;
	vpq_astExceptionListTable				: ARRAY[1..10] OF TPL.ST_Exception;
	vpiq_udiExceptionListGoToDetailsOfLine	: UDINT; (* index of the line that was selected in the exception list; set by vis to value, restet by VisControl; *)

	vpq_xShowExtendedTimes 					: BOOL := FALSE;
	vpq_xShowExtended2						: BOOL := FALSE;	
	vpiq_xButtonShowExtendedTimes 			: BOOL := FALSE;
	vpiq_xButtonShowExtended2				: BOOL := FALSE;
	
	vpq_udiNumberOfExceptions				: UDINT;
	
	udiIndex								: UDINT;
	vpq_sAllActiveReactions						: STRING[255];
	(* --- exception list --- *)

	udiExceptionListDetailsSelectIndex 		: UDINT;

	(*FR_ASCIILoggerList, navigation in the LoggerList*)
	vpiq_udiLogDataListIndexMin				: UDINT := 1;
	vpq_udiLogDataListIndexMax				: UDINT := 1;
	vpiq_udiNumberOfLogData					: UDINT;
	vpq_xLogDataScrollDown					: BOOL;
	vpq_astLogDataTableAscii				: ARRAY[1..12] OF TPL.ST_LogDataAscii;
	vpq_astLogDataTable						: ARRAY[1..12] OF TPL.ST_LogData;
	udiIndex2								: UDINT;
	udiIndex3								: UDINT;

	(*Variables to change color of the DiagQuit button*)
	vpq_dwDiagQuitColor					: DWORD;
	xRedColor							: BOOL;


	(* test exceptions *)
	stUserException1						: TPL.ST_Exception;
	stUserException2						: TPL.ST_Exception;
	stUserException3						: TPL.ST_Exception;
	stUserException4						: TPL.ST_Exception;
	stUserException5						: TPL.ST_Exception;

	(* copy of the ExceptionList *)
	fbCopyExceptionList						: TPL.FB_CopyExceptionList;
	astExceptionListCopy 					: ARRAY[1..TPL.Gc_udiMaxNumberOfExceptions] OF TPL.ST_Exception;
	
	vpiq_fbVisContExHandling					: TPL.FB_VisControllerExceptionHandling;

	(* Additional FBs for other types of modules *)
	vpiq_fbAxisModuleVisController : AXM.FB_AxisModuleVisController;
	(* For the RoboticModule *)
	//vpiq_fbRoboticModuleVisController : RM.FB_RoboticModuleVisController;

	(* For the ExampleLeafModule *)
	vpiq_fbExampleLeafModuleVisController : FB_ExampleLeafModuleVisController;


	fbDetectOnlineChange					: TPL.FB_DetectOnlineChange;
	xDetectOnlineChangeActive				: BOOL; 
	xDetectOnlineChangeReady				: BOOL; 
	etDetectOnlineChangeDiag				: GD.ET_Diag;
	etDetectOnlineChangeDiagExt				: TPL.ET_DiagExt; 
	sDetectOnlineChangeMsg					: STRING[80];
	xUpdatePointer							: BOOL;
	fbLoggerPoint							: APL.FB_LoggerPoint;
	
	(* Highlight the currently active OpMode (VIS_AxisModule) *)
	v_diLastOpMode							: DINT;
	v_xHomeModeActive						: BOOL;
	v_xManualModeActive						: BOOL;
	v_xMultiCamCSActive						: BOOL;
	v_xMultiCamWSActive						: BOOL;
	v_xEndlessActive						: BOOL;
	v_xEndlessILSActive						: BOOL;
	v_xPositioningActive					: BOOL;
	v_xBrakeActive							: BOOL;
	v_xAdditionalCSActive					: BOOL;
	v_xAdditionalWSActive					: BOOL;
END_VAR

(* Make sure that after an online-change, the main machine program has been executed
   before you update the pointers in the VisControl. *)
   
fbDetectOnlineChange(	i_xEnable	:= TRUE, 
						i_xDetect	:= TRUE, 
						q_xActive	=> xDetectOnlineChangeActive, 
						q_xReady	=> xDetectOnlineChangeReady, 
						q_etDiag	=> etDetectOnlineChangeDiag, 
						q_etDiagExt	=> etDetectOnlineChangeDiagExt, 
						q_sMsg		=> sDetectOnlineChangeMsg, 
						q_xChange	=> );
							
IF fbDetectOnlineChange.q_xChange THEN
	xUpdatePointer := TRUE;
	RETURN;
END_IF

IF G_xDoEnableVis THEN
	IF SR_MainMachine.stMachineInterface.q_xActive AND (iDoEnableCycleCounter < 3) THEN
		(* Wait until main machine ist active, otherwise some module vis
		controllers would read a wrong module structure. *)
		
		iDoEnableCycleCounter := iDoEnableCycleCounter + 1;
		IF iDoEnableCycleCounter >= 3 THEN
			(* This also assures, that all values and structures are initialized
			by the main machine when this task tries to access them. *)
			vpq_xDoEnable := TRUE;
		END_IF
	END_IF
ELSE
	vpq_xDoEnable := FALSE;
	
	iDoEnableCycleCounter := 0;
END_IF;

IF vpq_xDoEnable AND NOT xEnableFlag THEN
	xEnableFlag := TRUE;
	
	(* Initialize navigation *)
	pstCurrentParent			:= 0;
	pstCurrent					:= ADR(SR_MainMachine.stMachineInterface);
	udiCurrentLevel				:= 1;
	udiCurrentLevelSize			:= 1;
	audiHierarchy[1]			:= 1;
	xCurrentHasSubModules		:= (pstCurrent^.iq_stExt.udiNumberOfSubModules > 0);
	xCurrentHasControlModules	:= (pstCurrent^.iq_stExt.udiNumberOfControlModules > 0);
	xPointerExceptionActive		:= FALSE;
	xUpdateData					:= TRUE;
	udiMinModuleList			:= 1;
	udiMinSubModuleList			:= 1;
	udiCurrentLevel3Size		:= 0;
	vpiq_axModuleList			:= axClearBoolA5;
	vpiq_axSubModuleList			:= axClearBoolA5;

	udiCurrentNumberOfControlModules	:= 0;
	udiNumberOfControlModulesLevel2		:= 0;
	udiControlModuleSelectedInLevel		:= 0;
	vpq_udiActiveControlModuleNumber		:= 0;

	(* init test exceptions *)
	vpq_stMachineInterface := SR_MainMachine.stMachineInterface; (* required *)
	
	InitTestExceptions();

	vpq_xCurrentIsJogTarget := FALSE;
	
	fbLoggerPoint.RegisterLoggerPoint(	i_ifParent	:= APL.G_ifApplicationLogger,
										i_sName		:= 'VisControl',
										i_sType		:= 'SR_VisControl',
										i_sSource	:= 'Project',
										q_etDiag	=> ,
										q_etDiagExt	=> );
	iState := 10;
		
ELSIF NOT vpq_xDoEnable AND xEnableFlag THEN
	xEnableFlag := FALSE;
	
	G_xPrepareActive		:= FALSE;
	G_xAutoActive			:= FALSE;
	G_xManualActive			:= FALSE;
	G_xJogMachineActive		:= FALSE;
	G_xBrakeReleaseActive	:= FALSE;
	G_xTestMulticarrierActive	:= FALSE;
	
	iState := 5;
END_IF

CASE iState OF

0:
	iState := 5;

5:
	;

10:

	OpModeControl();

	(* Copy the machine interface into local variable, the local variable is read by the vis *)
	vpq_stMachineInterface := SR_MainMachine.stMachineInterface;

	vpq_xMachineInException := G_stExceptionList.udiNumberOfActiveExceptions > 0;

	vpq_etMainModuleControllerDiag		:= SR_MainMachine.fbModuleController.q_etDiag;
	vpq_etMainModuleControllerDiagExt	:= SR_MainMachine.fbModuleController.q_etDiagExt;
	vpq_sMainModuleControllerMsg			:= SR_MainMachine.fbModuleController.q_sMsg;

	MainPageCmdTable();
	
	ExceptionVis();

	LoggerVis();

	IF (G_xDiagQuitEpas AND xPointerExceptionActive) THEN
		xPointerExceptionActive := FALSE;
		
		udiCurrentLevel					:= 1;
		audiHierarchy[udiCurrentLevel]	:= 1;
		udiCurrentLevelSize				:= 1;
		xUpdateData						:= TRUE;
		vpiq_xButtonSetCurrentAsJogTarget			:= FALSE;
	END_IF

	IF (NOT xPointerExceptionActive) THEN

		ModuleNavigationIn();

		IF (xUpdateData OR xUpdatePointer) THEN
			xUpdateData		:= FALSE;
			xUpdatePointer	:= FALSE;
			
			xUpdateForOtherFBs := TRUE;

			(* Select current module *)
			SearchCurrentModule();

			ModuleNavigationOut();

		END_IF (* xUpdateData *)

		ModuleReaction();

		(* Cyclic reading of values from the structures *)
		IF pstCurrent <> 0 THEN (* Security check *)

			(* Execute user inputs first *)
			IF(vpiq_xEnableModuleClicked) THEN
				vpiq_xEnableModuleClicked := FALSE;
				pstCurrent^.i_xEnable := NOT pstCurrent^.i_xEnable;
			END_IF
			
			IF(vpiq_xSetCmdClicked) THEN
				vpiq_xSetCmdClicked := FALSE;
				pstCurrent^.iq_diCmd := vpiq_diCmdToSet;
				pstCurrent^.iq_diStartStep := vpiq_diStartStepToSet;
			END_IF
			
			IF(xDiagQuit_Touch) THEN
				xDiagQuit_WasTouched 		:= TRUE;
				pstCurrent^.i_xDiagQuit 	:= TRUE;
			ELSIF(xDiagQuit_WasTouched) THEN
				xDiagQuit_WasTouched 		:= FALSE;
				pstCurrent^.i_xDiagQuit 	:= FALSE;
			END_IF
			
			vpq_stCurrentModuleStandardInterface := pstCurrent^;


			(* If the current module is not selected as target for the jogForw, jogBack Buttons *)
			vpq_xCurrentIsJogTarget := (vpq_stCurrentModuleStandardInterface.i_udiModuleId = SR_MainMachine.stMachineMotionInterface.i_udiModuleSelect);
			
			(* this detects a change of the current module ==> the user has navigated to a different module.
				To avoid that the old and no longer visible module is jogged further, delete the jog target *)
			IFB_FTrigxCurrentIsJogTarget(CLK:= vpq_xCurrentIsJogTarget );
			IF IFB_FTrigxCurrentIsJogTarget.Q THEN
				G_udiManualModuleSelect := 0;	(*No Module can be jogged unintentionally*)
			END_IF

		ELSE
			vpq_stCurrentModuleStandardInterface	:= stDummyStandardInterface;
			udiCurrentLevelSize					:= 0;
			xCurrentHasSubModules				:= FALSE;
			udiCurrentLevel						:= 1;
			xUpdateData							:= TRUE;
			vpq_xCurrentIsJogTarget					:= FALSE;
		END_IF

		IF pstCurrentControlModuleStandardInterface <> 0 AND vpq_udiActiveControlModuleNumber > 0 THEN
			pstTempCtrlModule := pstCurrentControlModuleStandardInterface +  UDINT_TO_DWORD((vpq_udiActiveControlModuleNumber-1) * SIZEOF(pstCurrentControlModuleStandardInterface^));
			stCurrentControlModuleStandardInterface := pstTempCtrlModule^;
		ELSE
			stCurrentControlModuleStandardInterface.udiControlModuleNumber			:= 0;
			stCurrentControlModuleStandardInterface.udiControlModuleType			:= 0;
			stCurrentControlModuleStandardInterface.dwControlModuleAddItf			:= 0;
			stCurrentControlModuleStandardInterface.sControlModuleName				:= '';
		END_IF

		vpq_xButtonSetJogTargetInvisible := NOT SR_MainMachine.xOutputManualActive;

		(* Select the current module as target for the jogging *)
		IF(SR_MainMachine.xOutputManualActive) THEN
			(* Check whether we are really in jog mode *)
			IF(vpiq_xButtonSetCurrentAsJogTarget) THEN
				G_udiManualModuleSelect := vpq_stCurrentModuleStandardInterface.i_udiModuleId;
			END_IF
		END_IF
		
		vpiq_xButtonSetCurrentAsJogTarget := FALSE;

		(* generate additional output for the frame FR_CurrentModule *)
		vpq_sCurrentModuleReaction := TPL.FC_ReactionToString(iq_stReaction := vpq_stCurrentModuleStandardInterface.i_stReaction);

		CurrentModuleCmdTable();
	END_IF(* xPointerExceptionActive *)
(****************************************************************************************************************************************************)
END_CASE

IF(NOT xPointerExceptionActive) THEN
	(* point to call additional visualization controllers *)

	(* from Vis_ActiveExceptionList to Vis_ExceptionDetails *)
	IF(vpiq_udiExceptionListGoToDetailsOfLine <> 0) THEN
		IF(vpiq_udiExceptionListGoToDetailsOfLine > 0 AND vpiq_udiExceptionListGoToDetailsOfLine <= 10) THEN
			udiExceptionListDetailsSelectIndex := vpiq_udiExceptionListIndexMin + vpiq_udiExceptionListGoToDetailsOfLine - 1;
		END_IF
		vpiq_udiExceptionListGoToDetailsOfLine := 0;
	END_IF
	
	(* exception handling *)
	vpiq_fbVisContExHandling(	i_xEnable							:= vpq_xDoEnable,
								i_pstMachineStandardItf				:= ADR(SR_MainMachine.stMachineInterface),
								i_pstCurrentStandardItf				:= pstCurrent,
								i_xUpdateData						:= xUpdateForOtherFBs,
								i_udiNumberOfExceptions				:= vpq_udiNumberOfExceptions,
								iq_stExceptionList					:= G_stExceptionList,
								iq_stLogDataList					:= G_stLogDataList,
								iq_astExceptionListCopy				:= astExceptionListCopy,
								iq_udiExceptionDetailsSelectIndex	:= udiExceptionListDetailsSelectIndex,
								q_udiSetAsCurrentModule				=> udiSetAsCurrentModule);
						
	SetCurrentModule();

	(* module specific vis controllers are called inside this action *)
	ModuleVisController();


	(* End of area for vis control fbs of different module types *)
	xUpdateForOtherFBs := FALSE;
END_IF

(* Detect change of OpMode for AxisModule *)
DetectOpModeChange();

ACTION CallTestErrors:
TPL.FC_SetException(i_xExceptionActive := vpiq_xTestUserException1,
					iq_stException := stUserException1,
					iq_stExceptionList := G_stExceptionList,
					iq_stLogDataList := G_stLogDataList);
IF vpiq_xTestUserException1 AND NOT xTestUserException1Old AND (fbLoggerPoint.etLogLevel >= APL.ET_LogLevel.Exception) THEN
	fbLoggerPoint.AddLogEntry(	i_etLogLevel	:= APL.ET_LogLevel.Exception,
								i_etDiag		:= stUserException1.etDiag,
								i_udiDiagExt	:= stUserException1.udiDiagExt,
								i_sMessage		:= stUserException1.sMsg,
								q_etDiag		=> ,
								q_etDiagExt		=> );
END_IF
xTestUserException1Old := vpiq_xTestUserException1; 
	
TPL.FC_SetException(i_xExceptionActive := vpiq_xTestUserException2,
					iq_stException := stUserException2,
					iq_stExceptionList := G_stExceptionList,
					iq_stLogDataList := G_stLogDataList);
IF vpiq_xTestUserException2 AND NOT xTestUserException2Old AND (fbLoggerPoint.etLogLevel >= APL.ET_LogLevel.Exception) THEN
	fbLoggerPoint.AddLogEntry(	i_etLogLevel	:= APL.ET_LogLevel.Exception,
								i_etDiag		:= stUserException2.etDiag,
								i_udiDiagExt	:= stUserException2.udiDiagExt,
								i_sMessage		:= stUserException2.sMsg,
								q_etDiag		=> ,
								q_etDiagExt		=> );
END_IF
xTestUserException2Old := vpiq_xTestUserException2;
	
TPL.FC_SetException(i_xExceptionActive := vpiq_xTestUserException3,
					iq_stException := stUserException3,
					iq_stExceptionList := G_stExceptionList,
					iq_stLogDataList := G_stLogDataList);
IF vpiq_xTestUserException3 AND NOT xTestUserException3Old AND (fbLoggerPoint.etLogLevel >= APL.ET_LogLevel.Exception) THEN
	fbLoggerPoint.AddLogEntry(	i_etLogLevel	:= APL.ET_LogLevel.Exception,
								i_etDiag		:= stUserException3.etDiag,
								i_udiDiagExt	:= stUserException3.udiDiagExt,
								i_sMessage		:= stUserException3.sMsg,
								q_etDiag		=> ,
								q_etDiagExt		=> );
END_IF
xTestUserException3Old := vpiq_xTestUserException3;
	
TPL.FC_SetException(i_xExceptionActive := (vpiq_xTestUserException4 OR vpiq_fbAxisModuleVisController.q_xSimulateExceptionStopEndOfCycle),
					iq_stException := stUserException4,
					iq_stExceptionList := G_stExceptionList,
					iq_stLogDataList := G_stLogDataList);
IF (vpiq_xTestUserException4 OR vpiq_fbAxisModuleVisController.q_xSimulateExceptionStopEndOfCycle) AND NOT xTestUserException4Old AND (fbLoggerPoint.etLogLevel >= APL.ET_LogLevel.Exception) THEN
	fbLoggerPoint.AddLogEntry(	i_etLogLevel	:= APL.ET_LogLevel.Exception,
								i_etDiag		:= stUserException4.etDiag,
								i_udiDiagExt	:= stUserException4.udiDiagExt,
								i_sMessage		:= stUserException4.sMsg,
								q_etDiag		=> ,
								q_etDiagExt		=> );
END_IF
xTestUserException4Old := (vpiq_xTestUserException4 OR vpiq_fbAxisModuleVisController.q_xSimulateExceptionStopEndOfCycle);
	
TPL.FC_SetException(i_xExceptionActive := vpiq_xTestUserException5,
					iq_stException := stUserException5,
					iq_stExceptionList := G_stExceptionList,
					iq_stLogDataList := G_stLogDataList);
IF vpiq_xTestUserException5 AND NOT xTestUserException5Old AND (fbLoggerPoint.etLogLevel >= APL.ET_LogLevel.Exception) THEN
	fbLoggerPoint.AddLogEntry(	i_etLogLevel	:= APL.ET_LogLevel.Exception,
								i_etDiag		:= stUserException5.etDiag,
								i_udiDiagExt	:= stUserException5.udiDiagExt,
								i_sMessage		:= stUserException5.sMsg,
								q_etDiag		=> ,
								q_etDiagExt		=> );
END_IF
xTestUserException5Old := vpiq_xTestUserException5;
END_ACTION

ACTION CurrentModuleCmdTable:
(* Find the active CMD table *)
vpq_udiNumberOfCmdStepsModule :=  0; (* Default values, for security *)
pstEQCMDTableListEntry := 0;
pstEQCMDTable := 0;
IF (vpq_stCurrentModuleStandardInterface.q_diCMDActive <> 0 AND 
	vpq_stCurrentModuleStandardInterface.iq_stExt.udiNumberOfCMDTables > 0 AND 
	vpq_stCurrentModuleStandardInterface.iq_stExt.pstListofCMDTables <> 0) THEN
	
	FOR udiTmp2 := 1 TO vpq_stCurrentModuleStandardInterface.iq_stExt.udiNumberOfCMDTables DO
		pstEQCMDTableListEntry := vpq_stCurrentModuleStandardInterface.iq_stExt.pstListofCMDTables +  UDINT_TO_DWORD((udiTmp2-1)*SIZEOF(pstEQCMDTableListEntry^));
		IF(pstEQCMDTableListEntry^.diCMD = vpq_stCurrentModuleStandardInterface.q_diCMDActive) THEN (* Found *)
			vpq_udiNumberOfCmdStepsModule := pstEQCMDTableListEntry^.udiNumberOfCmdSteps;
			pstEQCMDTable := pstEQCMDTableListEntry^.pstCMDTable;
			vpq_sCmdTitleModule := pstEQCMDTableListEntry^.sTitle;
			EXIT;
		END_IF
	END_FOR
END_IF

(*Command steps > 10 and index changed??*)
IF vpq_udiNumberOfCmdStepsModule <> udiEQTableIndexOld OR udiEQTableStepCountOld <> vpq_udiNumberOfCmdStepsModule THEN
														(*More than 10 steps ??*)
	IF (vpiq_udiIndexMinModule + 9 < vpq_udiNumberOfCmdStepsModule) THEN
		udiEQTableIndexMax := vpiq_udiIndexMinModule + 9;
	ELSE
		udiEQTableIndexMax := vpq_udiNumberOfCmdStepsModule;
	END_IF
														(*Additional safety check*)
	IF (vpiq_udiIndexMinModule < 1) OR (vpiq_udiIndexMinModule > vpq_udiNumberOfCmdStepsModule) THEN
		vpiq_udiIndexMinModule :=1;
		udiEQTableIndexMax := 10;
	END_IF

	udiEQTableIndexOld := vpiq_udiIndexMinModule;
	udiEQTableStepCountOld := vpq_udiNumberOfCmdStepsModule;
END_IF (*vpiq_udiIndexMinModule <> udiEQTableIndexOld*)

vpq_xDisableScrollUpModule := NOT (vpiq_udiIndexMinModule > 1);
vpq_xDisableScrollDownModule := NOT (vpiq_udiIndexMinModule + 9 < vpq_udiNumberOfCmdStepsModule);

IF(pstEQCMDTable <> 0) THEN
	FOR udiCounter := udiEQTableIndexOld TO udiEQTableIndexMax DO
		pstEQCMDTableEntry := pstEQCMDTable +  UDINT_TO_DWORD(((udiCounter-1) * SIZEOF(pstEQCMDTable^)));
		vpq_astActualCmdTableModule[udiCounter - udiEQTableIndexOld + 1] := pstEQCMDTableEntry^;
	END_FOR
	FOR udiCounter := udiEQTableIndexMax + 1 TO udiEQTableIndexOld + 9 DO
		vpq_astActualCmdTableModule[udiCounter - udiEQTableIndexOld + 1] := c_stEmptyCmdTableStep;
	END_FOR
	vpq_xDisplayCmdTable := TRUE;
ELSE
	vpq_xDisplayCmdTable := FALSE;
END_IF
END_ACTION

ACTION DetectOpModeChange:
IF (vpiq_fbAxisModuleVisController.i_pstCurrentStandardItf <> 0) THEN
	IF (v_diLastOpMode <> vpiq_fbAxisModuleVisController.i_pstCurrentStandardItf^.q_diCmdActive) THEN
		v_diLastOpMode := vpiq_fbAxisModuleVisController.i_pstCurrentStandardItf^.q_diCmdActive;
		CASE (v_diLastOpMode) OF
			AXM.ET_Cmd.Homing:
				v_xHomeModeActive := TRUE;
				v_xManualModeActive := FALSE;
				v_xMultiCamCSActive := FALSE;
				v_xMultiCamWSActive := FALSE;
				v_xEndlessActive := FALSE;
				v_xEndlessILSActive := FALSE;
				v_xPositioningActive := FALSE;
				v_xBrakeActive := FALSE;
				v_xAdditionalCSActive := FALSE;
				v_xAdditionalWSActive := FALSE;		
			AXM.ET_Cmd.Manual:
				v_xHomeModeActive := FALSE;
				v_xManualModeActive := TRUE;
				v_xMultiCamCSActive := FALSE;
				v_xMultiCamWSActive := FALSE;
				v_xEndlessActive := FALSE;
				v_xEndlessILSActive := FALSE;
				v_xPositioningActive := FALSE;
				v_xBrakeActive := FALSE;
				v_xAdditionalCSActive := FALSE;
				v_xAdditionalWSActive := FALSE;
			
			AXM.ET_Cmd.CamCs:
				v_xHomeModeActive := FALSE;
				v_xManualModeActive := FALSE;
				v_xMultiCamCSActive := TRUE;
				v_xMultiCamWSActive := FALSE;
				v_xEndlessActive := FALSE;
				v_xEndlessILSActive := FALSE;
				v_xPositioningActive := FALSE;
				v_xBrakeActive := FALSE;
				v_xAdditionalCSActive := FALSE;
				v_xAdditionalWSActive := FALSE;
			
			AXM.ET_Cmd.CamWs:
				v_xHomeModeActive := FALSE;
				v_xManualModeActive := FALSE;
				v_xMultiCamCSActive := FALSE;
				v_xMultiCamWSActive := TRUE;
				v_xEndlessActive := FALSE;
				v_xEndlessILSActive := FALSE;
				v_xPositioningActive := FALSE;
				v_xBrakeActive := FALSE;
				v_xAdditionalCSActive := FALSE;
				v_xAdditionalWSActive := FALSE;
			
			AXM.ET_Cmd.Endless:
				v_xHomeModeActive := FALSE;
				v_xManualModeActive := FALSE;
				v_xMultiCamCSActive := FALSE;
				v_xMultiCamWSActive := FALSE;
				v_xEndlessActive := TRUE;
				v_xEndlessILSActive := FALSE;
				v_xPositioningActive := FALSE;
				v_xBrakeActive := FALSE;
				v_xAdditionalCSActive := FALSE;
				v_xAdditionalWSActive := FALSE;
			
			AXM.ET_Cmd.EndlessIls:
				v_xHomeModeActive := FALSE;
				v_xManualModeActive := FALSE;
				v_xMultiCamCSActive := FALSE;
				v_xMultiCamWSActive := FALSE;
				v_xEndlessActive := FALSE;
				v_xEndlessILSActive := TRUE;
				v_xPositioningActive := FALSE;
				v_xBrakeActive := FALSE;
				v_xAdditionalCSActive := FALSE;
				v_xAdditionalWSActive := FALSE;
			
			AXM.ET_Cmd.Positioning:
				v_xHomeModeActive := FALSE;
				v_xManualModeActive := FALSE;
				v_xMultiCamCSActive := FALSE;
				v_xMultiCamWSActive := FALSE;
				v_xEndlessActive := FALSE;
				v_xEndlessILSActive := FALSE;
				v_xPositioningActive := TRUE;
				v_xBrakeActive := FALSE;
				v_xAdditionalCSActive := FALSE;
				v_xAdditionalWSActive := FALSE;
			
			AXM.ET_Cmd.BrakeRelease:
				v_xHomeModeActive := FALSE;
				v_xManualModeActive := FALSE;
				v_xMultiCamCSActive := FALSE;
				v_xMultiCamWSActive := FALSE;
				v_xEndlessActive := FALSE;
				v_xEndlessILSActive := FALSE;
				v_xPositioningActive := FALSE;
				v_xBrakeActive := TRUE;
				v_xAdditionalCSActive := FALSE;
				v_xAdditionalWSActive := FALSE;
			
			AXM.ET_Cmd.AdditionalCs:
				v_xHomeModeActive := FALSE;
				v_xManualModeActive := FALSE;
				v_xMultiCamCSActive := FALSE;
				v_xMultiCamWSActive := FALSE;
				v_xEndlessActive := FALSE;
				v_xEndlessILSActive := FALSE;
				v_xPositioningActive := FALSE;
				v_xBrakeActive := FALSE;
				v_xAdditionalCSActive := TRUE;
				v_xAdditionalWSActive := FALSE;
			
			AXM.ET_Cmd.AdditionalWs:
				v_xHomeModeActive := FALSE;
				v_xManualModeActive := FALSE;
				v_xMultiCamCSActive := FALSE;
				v_xMultiCamWSActive := FALSE;
				v_xEndlessActive := FALSE;
				v_xEndlessILSActive := FALSE;
				v_xPositioningActive := FALSE;
				v_xBrakeActive := FALSE;
				v_xAdditionalCSActive := FALSE;
				v_xAdditionalWSActive := TRUE;
		END_CASE
	END_IF
END_IF
END_ACTION

ACTION ExceptionVis:
stActiveReactions := vpq_stMachineInterface.i_stReaction;

fbCopyExceptionList(i_xEnable					:= TRUE,
					i_xCopy						:= TRUE,
					i_timElapsedTimeUpdate		:= T#1S, (* update todElapsedTime every seccond, is fast enough for user interface *)
					iq_stExceptionList			:= G_stExceptionList,
					iq_astException				:= astExceptionListCopy,
					iq_udiNumberOfExceptions	:= vpq_udiNumberOfExceptions,
					q_xActive					=> ,
					q_xReady					=> ,
					q_etDiag					=> ,
					q_etDiagExt					=> );

IF vpiq_xReactionUp THEN
	vpq_udiReactionIndexMin := vpq_udiReactionIndexMin + 1;
	vpiq_xReactionUp:=FALSE;
ELSIF vpiq_xReactionDown THEN
	vpq_udiReactionIndexMin := vpq_udiReactionIndexMin - 1;
	vpiq_xReactionDown:=FALSE;
END_IF

IF vpq_udiReactionIndexMin <> udiReactionIndexOld THEN
														(*More than 10 steps ??*)
	IF (vpq_udiReactionIndexMin + 9 < TPL.Gc_udiMaxNumberOfReactions) THEN
		udiReactionIndexMax := vpq_udiReactionIndexMin + 9;
	ELSE
		udiReactionIndexMax := TPL.Gc_udiMaxNumberOfReactions;
	END_IF
														(*Additional safety check*)
	IF (vpq_udiReactionIndexMin < 1) THEN
		vpq_udiReactionIndexMin := 1;
		udiReactionIndexMax := 10;
	ELSIF (vpq_udiReactionIndexMin > TPL.Gc_udiMaxNumberOfReactions - 9) THEN
		vpq_udiReactionIndexMin := TPL.Gc_udiMaxNumberOfReactions - 9;
		udiReactionIndexMax := 10;
	END_IF

	udiReactionIndexOld := vpq_udiReactionIndexMin;
END_IF

IF TPL.Gc_udiMaxNumberOfReactions < 10 THEN
	udiMaxValue := TPL.Gc_udiMaxNumberOfReactions;
ELSE
	udiMaxValue := 10;
END_IF

FOR udiCount := 1 TO udiMaxValue  DO
	vpq_axReaction[udiCount] := stActiveReactions.axReaction[vpq_udiReactionIndexMin + udiCount - 1];
END_FOR

(*For Displaying the ErrorList-Visualization Vis_ActiveErrorList*)
IF vpiq_udiExceptionListIndexMin < 1 THEN
	vpiq_udiExceptionListIndexMin := 1;
END_IF

IF vpiq_udiExceptionListIndexMin > TPL.Gc_udiMaxNumberOfExceptions - 9 THEN
	vpiq_udiExceptionListIndexMin := TPL.Gc_udiMaxNumberOfExceptions - 9;
END_IF


FOR udiIndex := 1 TO 10 DO
	vpq_astExceptionListTable[udiIndex] := astExceptionListCopy[vpiq_udiExceptionListIndexMin + udiIndex - 1];
	vpq_asReaction [udiIndex] := TPL.FC_ReactionToString(astExceptionListCopy[vpiq_udiExceptionListIndexMin + udiIndex - 1].stReaction);
END_FOR

vpq_udiExceptionListIndexMax := vpiq_udiExceptionListIndexMin + 9;

IF vpq_udiExceptionListIndexMax > vpq_udiNumberOfExceptions - 1  THEN
	vpq_xDisplayScrollDown := TRUE;
ELSE
	vpq_xDisplayScrollDown := FALSE;
END_IF


vpq_sAllActiveReactions:= TPL.FC_ReactionToString(stActiveReactions);
CallTestErrors();

FOR udiCount := 1 TO TPL.Gc_udiMaxNumberOfReactions DO
	IF stActiveReactions.axReaction[udiCount] THEN
		xRedColor	:= TRUE;
		EXIT;
	ELSE
		xRedColor	:= FALSE;
	END_IF
END_FOR

IF xRedColor THEN
	vpq_dwDiagQuitColor := 16#FF0000;
ELSE
	vpq_dwDiagQuitColor := 16#FFFF00;
END_IF

IF vpiq_xButtonShowExtendedTimes AND NOT vpq_xShowExtendedTimes THEN
	vpq_xShowExtendedTimes		:= TRUE;
	vpq_xShowExtended2			:= FALSE;
	vpiq_xButtonShowExtendedTimes := FALSE;
	vpiq_xButtonShowExtended2		:= FALSE;
ELSIF vpiq_xButtonShowExtendedTimes  AND vpq_xShowExtendedTimes THEN
	vpq_xShowExtendedTimes		:= FALSE;
	vpq_xShowExtended2			:= FALSE;
	vpiq_xButtonShowExtendedTimes := FALSE;
	vpiq_xButtonShowExtended2		:= FALSE;
END_IF

IF vpiq_xButtonShowExtended2 AND NOT vpq_xShowExtended2 THEN
	vpq_xShowExtendedTimes		:= FALSE;
	vpq_xShowExtended2			:= TRUE;
	vpiq_xButtonShowExtendedTimes := FALSE;
	vpiq_xButtonShowExtended2		:= FALSE;
ELSIF vpiq_xButtonShowExtended2 AND vpq_xShowExtended2 THEN
	vpq_xShowExtendedTimes		:= FALSE;
	vpq_xShowExtended2			:= FALSE;
	vpiq_xButtonShowExtendedTimes := FALSE;
	vpiq_xButtonShowExtended2		:= FALSE;
END_IF
END_ACTION

ACTION InitTestExceptions:
stUserException1.etDiag														:= GD.ET_Diag.ExecutionAborted;
stUserException1.udiDiagExt													:= ET_DiagExt.Exception1FromVis;
stUserException1.sDiagExt													:= FC_EtDiagExtToString(ET_DiagExt.Exception1FromVis);
stUserException1.sMsg														:= 'Test Exception 1 from visualization - TPL.ET_Reaction.AsyncStop';
stUserException1.udiModuleId												:= vpq_stMachineInterface.i_udiModuleId;
stUserException1.sModuleName												:= vpq_stMachineInterface.i_sModuleName;
stUserException1.etSource													:= TPL.ET_ExceptionSource.Vis;
stUserException1.timDelayTime												:= T#0MS;
stUserException1.wHmiAttributes												:= 0;
stUserException1.xAutoQuit													:= FALSE;
stUserException1.stReaction.axReaction[TPL.ET_Reaction.AsyncStop]			:= TRUE;

